# B&R Automation Studio project NAEUL004C00R13L518F00 (part 17)

#### Act_OptP0928MagConv1BtmFB.st
```iecst
ACTION Act_OptP0928MagConv1BtmFB:

	//Magazine Conveyor
	IF tyP0928MagConv.tyBtmFB.tyBtnStop.bRtCompl = TRUE THEN
		eOutMagConvAct	:= MagConvActStop;

		IF p_eOutMagConvStat = MagConvActStop AND p_eOutMagConvStatus = Done THEN
			eOutMagConvAct	:= MagConvActIdle;

			tyP0928MagConv.tyBtmFB.tyBtnEnt.bRtCompl	:= FALSE;
			tyP0928MagConv.tyBtmFB.tyBtnEnt.bValue		:= FALSE;
			tyP0928MagConv.tyBtmFB.tyBtnEnt.bRtLk		:= FALSE;

			tyP0928MagConv.tyBtmFB.tyBtnExit.bRtCompl	:= FALSE;
			tyP0928MagConv.tyBtmFB.tyBtnExit.bValue		:= FALSE;
			tyP0928MagConv.tyBtmFB.tyBtnExit.bRtLk		:= FALSE;

			tyP0928MagConv.tyBtmFB.tyBtnStop.bRtCompl	:= FALSE;
			tyP0928MagConv.tyBtmFB.tyBtnStop.bValue		:= TRUE;
			tyP0928MagConv.tyBtmFB.tyBtnStop.bRtLk		:= TRUE;
		END_IF

	ELSIF tyP0928MagConv.tyBtmFB.tyBtnEnt.bRtCompl = TRUE THEN
		tyP0928MagConv.tyBtmFB.tyBtnEnt.bValue	:= TRUE;
		tyP0928MagConv.tyBtmFB.tyBtnEnt.bRtLk		:= TRUE;

		tyP0928MagConv.tyBtmFB.tyBtnStop.bValue	:= FALSE;
		tyP0928MagConv.tyBtmFB.tyBtnStop.bRtLk	:= FALSE;

		eOutMagConvAct	:= MagConvActEnt;

		IF p_eOutMagConvStat = MagConvActEnt AND p_eOutMagConvStatus = Done THEN
			eOutMagConvAct	:= MagConvActIdle;

			tyP0928MagConv.tyBtmFB.tyBtnEnt.bRtCompl	:= FALSE;

			tyP0928MagConv.tyBtmFB.tyBtnEnt.bValue	:= FALSE;
			tyP0928MagConv.tyBtmFB.tyBtnEnt.bRtLk		:= FALSE;

			tyP0928MagConv.tyBtmFB.tyBtnStop.bValue	:= TRUE;
			tyP0928MagConv.tyBtmFB.tyBtnStop.bRtLk	:= TRUE;
		END_IF

	ELSIF tyP0928MagConv.tyBtmFB.tyBtnExit.bRtCompl = TRUE THEN
		tyP0928MagConv.tyBtmFB.tyBtnExit.bValue	:= TRUE;
		tyP0928MagConv.tyBtmFB.tyBtnExit.bRtLk	:= TRUE;

		tyP0928MagConv.tyBtmFB.tyBtnStop.bValue	:= FALSE;
		tyP0928MagConv.tyBtmFB.tyBtnStop.bRtLk	:= FALSE;

		eOutMagConvAct	:= MagConvActExit;

		IF p_eOutMagConvStat = MagConvActExit AND p_eOutMagConvStatus = Done THEN
			eOutMagConvAct	:= MagConvActIdle;

			tyP0928MagConv.tyBtmFB.tyBtnExit.bRtCompl:= FALSE;

			tyP0928MagConv.tyBtmFB.tyBtnExit.bValue	:= FALSE;
			tyP0928MagConv.tyBtmFB.tyBtnExit.bRtLk	:= FALSE;

			tyP0928MagConv.tyBtmFB.tyBtnStop.bValue	:= TRUE;
			tyP0928MagConv.tyBtmFB.tyBtnStop.bRtLk	:= TRUE;
		END_IF
	END_IF

	//Stopper
	IF tyP0928MagConv.tyCom.tyBtnSwitch.bValue = FALSE THEN

		//Mid stopper
		IF tyP0928MagConv.tyBtmFB.tyBtnMidStprExt.bRtCompl = TRUE THEN
			tyP0928MagConv.tyBtmFB.tyBtnMidStprExt.bRtCompl	:= FALSE;

			tyP0928MagConv.tyBtmFB.tyBtnMidStprExt.bValue	:= TRUE;
			tyP0928MagConv.tyBtmFB.tyBtnMidStprRet.bValue	:= FALSE;

		ELSIF tyP0928MagConv.tyBtmFB.tyBtnMidStprRet.bRtCompl = TRUE THEN
			tyP0928MagConv.tyBtmFB.tyBtnMidStprRet.bRtCompl	:= FALSE;

			tyP0928MagConv.tyBtmFB.tyBtnMidStprRet.bValue	:= TRUE;
			tyP0928MagConv.tyBtmFB.tyBtnMidStprExt.bValue	:= FALSE;

		END_IF

		//Ext Stopper
		IF tyP0928MagConv.tyBtmFB.tyBtnExtStprExt.bRtCompl = TRUE THEN
			tyP0928MagConv.tyBtmFB.tyBtnExtStprExt.bRtCompl	:= FALSE;

			tyP0928MagConv.tyBtmFB.tyBtnExtStprExt.bValue	:= TRUE;
			tyP0928MagConv.tyBtmFB.tyBtnExtStprRet.bValue	:= FALSE;

		ELSIF tyP0928MagConv.tyBtmFB.tyBtnExtStprRet.bRtCompl = TRUE THEN
			tyP0928MagConv.tyBtmFB.tyBtnExtStprRet.bRtCompl	:= FALSE;

			tyP0928MagConv.tyBtmFB.tyBtnExtStprRet.bValue	:= TRUE;
			tyP0928MagConv.tyBtmFB.tyBtnExtStprExt.bValue	:= FALSE;

		END_IF

		//Action------------

		IF tyP0928MagConv.tyBtmFB.tyBtnMidStprExt.bValue = TRUE THEN
				eStopper4Act	:= PneuActExt;

				IF p_eStopper4Stat = PneuActExt AND p_eStopper4Status = Done THEN
					eStopper4Act	:= PneuActIdle;
					tyP0928MagConv.tyBtmFB.tyBtnMidStprExt.bValue	:= FALSE;
				ELSIF p_eStopper4Status = Error THEN
					tyP0928MagConv.tyBtmFB.tyBtnMidStprExt.bValue	:= FALSE;
				END_IF

		ELSIF tyP0928MagConv.tyBtmFB.tyBtnMidStprRet.bValue = TRUE THEN
			eStopper4Act	:= PneuActRet;

			IF p_eStopper4Stat = PneuActRet AND p_eStopper4Status = Done THEN
				eStopper4Act	:= PneuActIdle;
				tyP0928MagConv.tyBtmFB.tyBtnMidStprRet.bValue := FALSE;
			ELSIF p_eStopper4Status = Error THEN
				tyP0928MagConv.tyBtmFB.tyBtnMidStprRet.bValue := FALSE;
			END_IF

		END_IF

		IF tyP0928MagConv.tyBtmFB.tyBtnExtStprExt.bValue = TRUE THEN
			eStopper5Act	:= PneuActExt;

			IF p_eStopper5Stat = PneuActExt AND p_eStopper5Status = Done THEN
				eStopper5Act	:= PneuActIdle;
				tyP0928MagConv.tyBtmFB.tyBtnExtStprExt.bValue	:= FALSE;
			ELSIF p_eStopper5Status = Error THEN
				tyP0928MagConv.tyBtmFB.tyBtnExtStprExt.bValue	:= FALSE;
			END_IF

		ELSIF tyP0928MagConv.tyBtmFB.tyBtnExtStprRet.bValue = TRUE THEN
			eStopper5Act	:= PneuActRet;

			IF p_eStopper5Stat = PneuActRet AND p_eStopper5Status = Done THEN
				eStopper5Act	:= PneuActIdle;
				tyP0928MagConv.tyBtmFB.tyBtnExtStprRet.bValue := FALSE;
			ELSIF p_eStopper5Status = Error THEN
				tyP0928MagConv.tyBtmFB.tyBtnExtStprRet.bValue := FALSE;
			END_IF

		END_IF

		//Update Status
//		tyP0930MagConvBtm1.tyDC.tyBtnFixedUnclamp.bValue	:= NOT p_bMagConvBtm2Clp1ClprFixClampCtrl;
//		tyP0930MagConvBtm1.tyDC.tyBtnFixedClamp.bValue		:= p_bMagConvBtm2Clp1ClprFixClampCtrl;
//		tyP0930MagConvBtm1.tyDC.tyBtnRemoteUnclamp.bValue	:= NOT p_bMagConvBtm2Clp1ClprRmtClampCtrl;
//		tyP0930MagConvBtm1.tyDC.tyBtnRemoteClamp.bValue	:= p_bMagConvBtm2Clp1ClprRmtClampCtrl;
//
//		tyP0930MagConvBtm1.tyDC.tyBtnSelUnclamp.bRtCompl	:= FALSE;
//		tyP0930MagConvBtm1.tyDC.tyBtnSelClamp.bRtCompl		:= FALSE;
//		tyP0930MagConvBtm1.tyDC.tyBtnSelUnclamp.bValue	:= p_bSelClamp1RetCtrl;
//		tyP0930MagConvBtm1.tyDC.tyBtnSelClamp.bValue	:= p_bSelClamp1ExtCtrl;
	END_IF

	//Mask
//	IF p_tyUsrMgmtCurrAccessRgt.bManualFBOnly THEN
//
//		fUIInRtStatOff(ADR(tyP0930MagConvBtm1.tyCom.tyBtnSwitch.uiMaskRtStat));
//
//	ELSE
//
//	IF p_eMagConvBtm2Clp1Status = Error THEN
//
//		fUIInRtStatOff(ADR(tyP0930MagConvBtm1.tyFB.tyBtnEnt.uiMaskRtStat));
//		fUIInRtStatOff(ADR(tyP0930MagConvBtm1.tyFB.tyBtnExit.uiMaskRtStat));
//		fUIInRtStatOff(ADR(tyP0930MagConvBtm1.tyFB.tyBtnFixedClamp.uiMaskRtStat));
//		fUIInRtStatOff(ADR(tyP0930MagConvBtm1.tyFB.tyBtnFixedUnclamp.uiMaskRtStat));
//		fUIInRtStatOff(ADR(tyP0930MagConvBtm1.tyFB.tyBtnRemoteClamp.uiMaskRtStat));
//		fUIInRtStatOff(ADR(tyP0930MagConvBtm1.tyFB.tyBtnRemoteUnclamp.uiMaskRtStat));
//		fUIInRtStatOff(ADR(tyP0930MagConvBtm1.tyFB.tyBtnSelClamp.uiMaskRtStat));
//		fUIInRtStatOff(ADR(tyP0930MagConvBtm1.tyFB.tyBtnSelUnclamp.uiMaskRtStat));
//		fUIInRtStatHide(ADR(tyP0930MagConvBtm1.tyCom.tyBtnSwitch.uiMaskRtStat));
//
//	ELSIF tyP0930MagConvBtm1.tyFB.tyBtnEnt.bRtCompl = TRUE THEN
//
//		fUIInRtStatHide(ADR(tyP0930MagConvBtm1.tyFB.tyBtnEnt.uiMaskRtStat));
//		fUIInRtStatOff(ADR(tyP0930MagConvBtm1.tyFB.tyBtnExit.uiMaskRtStat));
//		fUIInRtStatOff(ADR(tyP0930MagConvBtm1.tyFB.tyBtnFixedClamp.uiMaskRtStat));
//		fUIInRtStatOff(ADR(tyP0930MagConvBtm1.tyFB.tyBtnFixedUnclamp.uiMaskRtStat));
//		fUIInRtStatOff(ADR(tyP0930MagConvBtm1.tyFB.tyBtnRemoteClamp.uiMaskRtStat));
//		fUIInRtStatOff(ADR(tyP0930MagConvBtm1.tyFB.tyBtnRemoteUnclamp.uiMaskRtStat));
//		fUIInRtStatOff(ADR(tyP0930MagConvBtm1.tyFB.tyBtnSelClamp.uiMaskRtStat));
//		fUIInRtStatOff(ADR(tyP0930MagConvBtm1.tyFB.tyBtnSelUnclamp.uiMaskRtStat));
//		fUIInRtStatOff(ADR(tyP0930MagConvBtm1.tyCom.tyBtnSwitch.uiMaskRtStat));
//
//	ELSIF tyP0930MagConvBtm1.tyFB.tyBtnExit.bRtCompl = TRUE THEN
//
//			fUIInRtStatOff(ADR(tyP0930MagConvBtm1.tyFB.tyBtnEnt.uiMaskRtStat));
//		fUIInRtStatHide(ADR(tyP0930MagConvBtm1.tyFB.tyBtnExit.uiMaskRtStat));
//		fUIInRtStatOff(ADR(tyP0930MagConvBtm1.tyFB.tyBtnFixedClamp.uiMaskRtStat));
//		fUIInRtStatOff(ADR(tyP0930MagConvBtm1.tyFB.tyBtnFixedUnclamp.uiMaskRtStat));
//		fUIInRtStatOff(ADR(tyP0930MagConvBtm1.tyFB.tyBtnRemoteClamp.uiMaskRtStat));
//		fUIInRtStatOff(ADR(tyP0930MagConvBtm1.tyFB.tyBtnRemoteUnclamp.uiMaskRtStat));
//		fUIInRtStatOff(ADR(tyP0930MagConvBtm1.tyFB.tyBtnSelClamp.uiMaskRtStat));
//		fUIInRtStatOff(ADR(tyP0930MagConvBtm1.tyFB.tyBtnSelUnclamp.uiMaskRtStat));
//		fUIInRtStatOff(ADR(tyP0930MagConvBtm1.tyCom.tyBtnSwitch.uiMaskRtStat));
//
//	ELSIF tyP0930MagConvBtm1.tyFB.tyBtnFixedClamp.bValue = TRUE OR tyP0930MagConvBtm1.tyFB.tyBtnRemoteClamp.bValue = TRUE
//			OR tyP0930MagConvBtm1.tyFB.tyBtnFixedUnclamp.bValue = TRUE OR tyP0930MagConvBtm1.tyFB.tyBtnRemoteUnclamp.bValue = TRUE
//			OR tyP0930MagConvBtm1.tyFB.tyBtnSelUnclamp.bValue = TRUE OR tyP0930MagConvBtm1.tyFB.tyBtnSelClamp.bValue = TRUE
//			THEN
//
//		fUIInRtStatOff(ADR(tyP0930MagConvBtm1.tyFB.tyBtnEnt.uiMaskRtStat));
//		fUIInRtStatOff(ADR(tyP0930MagConvBtm1.tyFB.tyBtnExit.uiMaskRtStat));
//		fUIInRtStatHide(ADR(tyP0930MagConvBtm1.tyFB.tyBtnFixedClamp.uiMaskRtStat));
//		fUIInRtStatHide(ADR(tyP0930MagConvBtm1.tyFB.tyBtnFixedUnclamp.uiMaskRtStat));
//		fUIInRtStatHide(ADR(tyP0930MagConvBtm1.tyFB.tyBtnRemoteClamp.uiMaskRtStat));
//		fUIInRtStatHide(ADR(tyP0930MagConvBtm1.tyFB.tyBtnRemoteUnclamp.uiMaskRtStat));
//		fUIInRtStatHide(ADR(tyP0930MagConvBtm1.tyFB.tyBtnSelClamp.uiMaskRtStat));
//		fUIInRtStatHide(ADR(tyP0930MagConvBtm1.tyFB.tyBtnSelUnclamp.uiMaskRtStat));
//		fUIInRtStatOff(ADR(tyP0930MagConvBtm1.tyCom.tyBtnSwitch.uiMaskRtStat));
//
//	ELSE
//
//		fUIInRtStatHide(ADR(tyP0930MagConvBtm1.tyFB.tyBtnEnt.uiMaskRtStat));
//		fUIInRtStatHide(ADR(tyP0930MagConvBtm1.tyFB.tyBtnExit.uiMaskRtStat));
//		fUIInRtStatHide(ADR(tyP0930MagConvBtm1.tyFB.tyBtnFixedClamp.uiMaskRtStat));
//		fUIInRtStatHide(ADR(tyP0930MagConvBtm1.tyFB.tyBtnFixedUnclamp.uiMaskRtStat));
//		fUIInRtStatHide(ADR(tyP0930MagConvBtm1.tyFB.tyBtnRemoteClamp.uiMaskRtStat));
//		fUIInRtStatHide(ADR(tyP0930MagConvBtm1.tyFB.tyBtnRemoteUnclamp.uiMaskRtStat));
//		fUIInRtStatHide(ADR(tyP0930MagConvBtm1.tyFB.tyBtnSelClamp.uiMaskRtStat));
//		fUIInRtStatHide(ADR(tyP0930MagConvBtm1.tyFB.tyBtnSelUnclamp.uiMaskRtStat));
//		fUIInRtStatHide(ADR(tyP0930MagConvBtm1.tyCom.tyBtnSwitch.uiMaskRtStat));
//
//	END_IF
//END_IF
//
//	IF p_tyDI.bMagConvBtmCAB717MagSen1 THEN
//			fUIInRtStatOff(ADR(tyP0930MagConvBtm1.tyFB.tyBtnSelClamp.uiMaskRtStat));
//	END_IF
//
//	IF p_bMagConvBtm2Clp1ClprFixClampCtrl OR p_bMagConvBtm2Clp1ClprRmtClampCtrl THEN
//		fUIInRtStatOff(ADR(tyP0930MagConvBtm1.tyFB.tyBtnEnt.uiMaskRtStat));
//		fUIInRtStatOff(ADR(tyP0930MagConvBtm1.tyFB.tyBtnExit.uiMaskRtStat));
//	END_IF
//

END_ACTION
```

#### Act_OptP0928MagConv1TopDC.st
```iecst
ACTION Act_OptP0928MagConv1TopDC:

	//Magazine Conveyor
	IF tyP0928MagConv.tyTopDC.tyBtnStop.bRtCompl = TRUE THEN
		eInMagConvAct	:= MagConvActStop;

		IF p_eInMagConvStat = MagConvActStop AND p_eInMagConvStatus = Done THEN
			eInMagConvAct	:= MagConvActIdle;

			tyP0928MagConv.tyTopDC.tyBtnStop.bRtCompl		:= FALSE;
			tyP0928MagConv.tyTopDC.tyBtnStop.bValue		:= TRUE;
			tyP0928MagConv.tyTopDC.tyBtnStop.bRtLk		:= TRUE;

			tyP0928MagConv.tyTopDC.tyBtnMagIn.bRtCompl	:= FALSE;
			tyP0928MagConv.tyTopDC.tyBtnMagIn.bValue		:= FALSE;
			tyP0928MagConv.tyTopDC.tyBtnMagIn.bRtLk		:= FALSE;

			tyP0928MagConv.tyTopDC.tyBtnMagOut.bRtCompl	:= FALSE;
			tyP0928MagConv.tyTopDC.tyBtnMagOut.bValue		:= FALSE;
			tyP0928MagConv.tyTopDC.tyBtnMagOut.bRtLk		:= FALSE;
		END_IF

	ELSIF tyP0928MagConv.tyTopDC.tyBtnMagIn.bRtCompl = TRUE THEN
		tyP0928MagConv.tyTopDC.tyBtnMagIn.bValue	:= TRUE;
		tyP0928MagConv.tyTopDC.tyBtnMagIn.bRtLk	:= TRUE;

		tyP0928MagConv.tyTopDC.tyBtnStop.bValue	:= FALSE;
		tyP0928MagConv.tyTopDC.tyBtnStop.bRtLk	:= FALSE;

		IF p_tyNtParamCurr.eProjInMagConvDir = ConvDirLToR OR p_tyNtParamCurr.eProjInMagConvDir = ConvDirLToL THEN

			eInMagConvAct	:= MagConvActSetMtrSigOnOrLToR;

			IF p_eInMagConvStat = MagConvActSetMtrSigOnOrLToR AND p_eInMagConvStatus = Done THEN
				eInMagConvAct	:= MagConvActIdle;

				tyP0928MagConv.tyTopDC.tyBtnMagIn.bRtCompl	:= FALSE;
			END_IF

		ELSE

			eInMagConvAct	:= MagConvActSetMtrDirOrRToL;

			IF p_eInMagConvStat = MagConvActSetMtrDirOrRToL AND p_eInMagConvStatus = Done THEN
				eInMagConvAct	:= MagConvActIdle;

				tyP0928MagConv.tyTopDC.tyBtnMagIn.bRtCompl	:= FALSE;
			END_IF

		END_IF

	ELSIF tyP0928MagConv.tyTopDC.tyBtnMagOut.bRtCompl = TRUE THEN
		tyP0928MagConv.tyTopDC.tyBtnMagOut.bValue	:= TRUE;
		tyP0928MagConv.tyTopDC.tyBtnMagOut.bRtLk	:= TRUE;

		tyP0928MagConv.tyTopDC.tyBtnStop.bValue	:= FALSE;
		tyP0928MagConv.tyTopDC.tyBtnStop.bRtLk	:= FALSE;

		IF p_tyNtParamCurr.eProjMagConvDir = ConvDirLToR OR p_tyNtParamCurr.eProjInMagConvDir = ConvDirRToR THEN

			eInMagConvAct	:= MagConvActSetMtrSigOnOrLToR;

			IF p_eInMagConvStat = MagConvActSetMtrSigOnOrLToR AND p_eInMagConvStatus = Done THEN
				eInMagConvAct	:= MagConvActIdle;

				tyP0928MagConv.tyTopDC.tyBtnMagOut.bRtCompl	:= FALSE;
			END_IF

		ELSE

			eInMagConvAct	:= MagConvActSetMtrDirOrRToL;

			IF p_eInMagConvStat = MagConvActSetMtrDirOrRToL AND p_eInMagConvStatus = Done THEN
				eInMagConvAct	:= MagConvActIdle;

				tyP0928MagConv.tyTopDC.tyBtnMagOut.bRtCompl	:= FALSE;
			END_IF

		END_IF

	END_IF

	IF tyP0928MagConv.tyCom.tyBtnSwitch.bValue = TRUE THEN
		//Mag Conv Stopper1
		IF p_bStopper1TwoCtrlOut = FALSE THEN
			IF tyP0928MagConv.tyTopDC.tyBtnEntStprExt.bRtCompl = TRUE THEN
				tyP0928MagConv.tyTopDC.tyBtnEntStprExt.bValue := TRUE;
				tyP0928MagConv.tyTopDC.tyBtnEntStprRet.bValue := FALSE;

				eStopper1Act	:= PneuActSetExt;

				IF p_eStopper1Stat = PneuActSetExt AND p_eStopper1Status = Done THEN
					eStopper1Act	:= PneuActIdle;

					tyP0928MagConv.tyTopDC.tyBtnEntStprExt.bRtCompl	:= FALSE;
				END_IF

			ELSIF tyP0928MagConv.tyTopDC.tyBtnEntStprRet.bRtCompl = TRUE THEN
				tyP0928MagConv.tyTopDC.tyBtnEntStprRet.bValue := TRUE;
				tyP0928MagConv.tyTopDC.tyBtnEntStprExt.bValue := FALSE;

				eStopper1Act	:= PneuActSetRet;

				IF p_eStopper1Stat = PneuActSetRet AND p_eStopper1Status = Done THEN
					eStopper1Act	:= PneuActIdle;

					tyP0928MagConv.tyTopDC.tyBtnEntStprRet.bRtCompl	:= FALSE;
				END_IF
			END_IF

		ELSE
			IF (tyP0928MagConv.tyTopDC.tyBtnEntStprExt.bRtCompl = TRUE) OR (tyP0928MagConv.tyTopDC.tyBtnEntStprRet.bRtCompl = TRUE) THEN
				IF (tyP0928MagConv.tyTopDC.tyBtnEntStprExt.bValue = TRUE) AND (tyP0928MagConv.tyTopDC.tyBtnEntStprRet.bValue = TRUE) THEN
					eStopper1Act	:= PneuActSetAll;

					IF p_eStopper1Stat = PneuActSetAll AND p_eStopper1Status = Done THEN
						eStopper1Act	:= PneuActIdle;

						tyP0928MagConv.tyTopDC.tyBtnEntStprExt.bRtCompl		:= FALSE;
						tyP0928MagConv.tyTopDC.tyBtnEntStprRet.bRtCompl			:= FALSE;
					END_IF
					/////////i edited the ret to ext
				ELSIF (tyP0928MagConv.tyTopDC.tyBtnEntStprExt.bValue = TRUE) AND (tyP0928MagConv.tyTopDC.tyBtnEntStprRet.bValue = FALSE) THEN
					eStopper1Act	:= PneuActSetExt;(**)

					IF p_eStopper1Stat = PneuActSetExt (**) AND p_eStopper1Status = Done THEN
						eStopper1Act	:= PneuActIdle;

						tyP0928MagConv.tyTopDC.tyBtnEntStprExt.bRtCompl		:= FALSE;
						tyP0928MagConv.tyTopDC.tyBtnEntStprRet.bRtCompl		:= FALSE;
					END_IF

				ELSIF (tyP0928MagConv.tyTopDC.tyBtnEntStprExt.bValue = FALSE) AND (tyP0928MagConv.tyTopDC.tyBtnEntStprRet.bValue = TRUE) THEN
					eStopper1Act	:= PneuActSetRet;

					IF p_eStopper1Stat = PneuActSetRet AND p_eStopper1Status = Done THEN
						eStopper1Act	:= PneuActIdle;

						tyP0928MagConv.tyTopDC.tyBtnEntStprExt.bRtCompl		:= FALSE;
						tyP0928MagConv.tyTopDC.tyBtnEntStprRet.bRtCompl			:= FALSE;
					END_IF
					///////
				ELSE
					eStopper1Act	:= PneuActRstAll;

					IF p_eStopper1Stat = PneuActRstAll AND p_eStopper1Status = Done THEN
						eStopper1Act	:= PneuActIdle;

						tyP0928MagConv.tyTopDC.tyBtnEntStprExt.bRtCompl		:= FALSE;
						tyP0928MagConv.tyTopDC.tyBtnEntStprRet.bRtCompl			:= FALSE;
					END_IF

				END_IF
			END_IF
		END_IF//stopper1

		//Mag Conv Stopper2
		IF p_bStopper2TwoCtrlOut = FALSE THEN
			IF tyP0928MagConv.tyTopDC.tyBtnMidStprExt.bRtCompl = TRUE THEN
				tyP0928MagConv.tyTopDC.tyBtnMidStprExt.bValue := TRUE;
				tyP0928MagConv.tyTopDC.tyBtnMidStprRet.bValue := FALSE;

				eStopper2Act	:= PneuActSetExt;

				IF p_eStopper2Stat = PneuActSetExt AND p_eStopper2Status = Done THEN
					eStopper2Act	:= PneuActIdle;

					tyP0928MagConv.tyTopDC.tyBtnMidStprExt.bRtCompl	:= FALSE;
				END_IF

			ELSIF tyP0928MagConv.tyTopDC.tyBtnMidStprRet.bRtCompl = TRUE THEN
				tyP0928MagConv.tyTopDC.tyBtnMidStprRet.bValue := TRUE;
				tyP0928MagConv.tyTopDC.tyBtnMidStprExt.bValue := FALSE;

				eStopper2Act	:= PneuActSetRet;

				IF p_eStopper2Stat = PneuActSetRet AND p_eStopper2Status = Done THEN
					eStopper2Act	:= PneuActIdle;

					tyP0928MagConv.tyTopDC.tyBtnMidStprRet.bRtCompl	:= FALSE;
				END_IF
			END_IF

		ELSE
			IF (tyP0928MagConv.tyTopDC.tyBtnMidStprExt.bRtCompl = TRUE) OR (tyP0928MagConv.tyTopDC.tyBtnMidStprRet.bRtCompl = TRUE) THEN
				IF (tyP0928MagConv.tyTopDC.tyBtnMidStprExt.bValue = TRUE) AND (tyP0928MagConv.tyTopDC.tyBtnMidStprRet.bValue = TRUE) THEN
					eStopper2Act	:= PneuActSetAll;

					IF p_eStopper2Stat = PneuActSetAll AND p_eStopper2Status = Done THEN
						eStopper2Act	:= PneuActIdle;

						tyP0928MagConv.tyTopDC.tyBtnMidStprExt.bRtCompl		:= FALSE;
						tyP0928MagConv.tyTopDC.tyBtnMidStprRet.bRtCompl			:= FALSE;
					END_IF
					/////////i edited the ret to ext
				ELSIF (tyP0928MagConv.tyTopDC.tyBtnMidStprExt.bValue = TRUE) AND (tyP0928MagConv.tyTopDC.tyBtnMidStprRet.bValue = FALSE) THEN
					eStopper2Act	:= PneuActSetExt;(**)

					IF p_eStopper2Stat = PneuActSetExt (**) AND p_eStopper2Status = Done THEN
						eStopper2Act	:= PneuActIdle;

						tyP0928MagConv.tyTopDC.tyBtnMidStprExt.bRtCompl		:= FALSE;
						tyP0928MagConv.tyTopDC.tyBtnMidStprRet.bRtCompl		:= FALSE;
					END_IF

				ELSIF (tyP0928MagConv.tyTopDC.tyBtnMidStprExt.bValue = FALSE) AND (tyP0928MagConv.tyTopDC.tyBtnMidStprRet.bValue = TRUE) THEN
					eStopper2Act	:= PneuActSetRet;

					IF p_eStopper2Stat = PneuActSetRet AND p_eStopper2Status = Done THEN
						eStopper2Act	:= PneuActIdle;

						tyP0928MagConv.tyTopDC.tyBtnMidStprExt.bRtCompl		:= FALSE;
						tyP0928MagConv.tyTopDC.tyBtnMidStprRet.bRtCompl			:= FALSE;
					END_IF
					///////
				ELSE
					eStopper2Act	:= PneuActRstAll;

					IF p_eStopper2Stat = PneuActRstAll AND p_eStopper2Status = Done THEN
						eStopper2Act	:= PneuActIdle;

						tyP0928MagConv.tyTopDC.tyBtnMidStprExt.bRtCompl		:= FALSE;
						tyP0928MagConv.tyTopDC.tyBtnMidStprRet.bRtCompl			:= FALSE;
					END_IF

				END_IF
			END_IF
		END_IF//stopper2

		//Mag Conv Stopper3
		IF p_bStopper3TwoCtrlOut = FALSE THEN
			IF tyP0928MagConv.tyTopDC.tyBtnExtStprExt.bRtCompl = TRUE THEN
				tyP0928MagConv.tyTopDC.tyBtnExtStprExt.bValue := TRUE;
				tyP0928MagConv.tyTopDC.tyBtnExtStprRet.bValue := FALSE;

				eStopper3Act	:= PneuActSetExt;

				IF p_eStopper3Stat = PneuActSetExt AND p_eStopper3Status = Done THEN
					eStopper3Act	:= PneuActIdle;

					tyP0928MagConv.tyTopDC.tyBtnExtStprExt.bRtCompl	:= FALSE;
				END_IF

			ELSIF tyP0928MagConv.tyTopDC.tyBtnExtStprRet.bRtCompl = TRUE THEN
				tyP0928MagConv.tyTopDC.tyBtnExtStprRet.bValue := TRUE;
				tyP0928MagConv.tyTopDC.tyBtnExtStprExt.bValue := FALSE;

				eStopper3Act	:= PneuActSetRet;

				IF p_eStopper3Stat = PneuActSetRet AND p_eStopper3Status = Done THEN
					eStopper3Act	:= PneuActIdle;

					tyP0928MagConv.tyTopDC.tyBtnExtStprRet.bRtCompl	:= FALSE;
				END_IF
			END_IF

		ELSE
			IF (tyP0928MagConv.tyTopDC.tyBtnExtStprExt.bRtCompl = TRUE) OR (tyP0928MagConv.tyTopDC.tyBtnExtStprRet.bRtCompl = TRUE) THEN
				IF (tyP0928MagConv.tyTopDC.tyBtnExtStprExt.bValue = TRUE) AND (tyP0928MagConv.tyTopDC.tyBtnExtStprRet.bValue = TRUE) THEN
					eStopper3Act	:= PneuActSetAll;

					IF p_eStopper3Stat = PneuActSetAll AND p_eStopper3Status = Done THEN
						eStopper3Act	:= PneuActIdle;

						tyP0928MagConv.tyTopDC.tyBtnExtStprExt.bRtCompl		:= FALSE;
						tyP0928MagConv.tyTopDC.tyBtnExtStprRet.bRtCompl			:= FALSE;
					END_IF
					/////////i edited the ret to ext
				ELSIF (tyP0928MagConv.tyTopDC.tyBtnExtStprExt.bValue = TRUE) AND (tyP0928MagConv.tyTopDC.tyBtnExtStprRet.bValue = FALSE) THEN
					eStopper3Act	:= PneuActSetExt;(**)

					IF p_eStopper3Stat = PneuActSetExt (**) AND p_eStopper3Status = Done THEN
						eStopper3Act	:= PneuActIdle;

						tyP0928MagConv.tyTopDC.tyBtnExtStprExt.bRtCompl		:= FALSE;
						tyP0928MagConv.tyTopDC.tyBtnExtStprRet.bRtCompl		:= FALSE;
					END_IF

				ELSIF (tyP0928MagConv.tyTopDC.tyBtnExtStprExt.bValue = FALSE) AND (tyP0928MagConv.tyTopDC.tyBtnExtStprRet.bValue = TRUE) THEN
					eStopper3Act	:= PneuActSetRet;

					IF p_eStopper3Stat = PneuActSetRet AND p_eStopper3Status = Done THEN
						eStopper3Act	:= PneuActIdle;

						tyP0928MagConv.tyTopDC.tyBtnExtStprExt.bRtCompl		:= FALSE;
						tyP0928MagConv.tyTopDC.tyBtnExtStprRet.bRtCompl			:= FALSE;
					END_IF
					///////
				ELSE
					eStopper3Act	:= PneuActRstAll;

					IF p_eStopper3Stat = PneuActRstAll AND p_eStopper3Status = Done THEN
						eStopper3Act	:= PneuActIdle;

						tyP0928MagConv.tyTopDC.tyBtnExtStprExt.bRtCompl		:= FALSE;
						tyP0928MagConv.tyTopDC.tyBtnExtStprRet.bRtCompl			:= FALSE;
					END_IF

				END_IF
			END_IF
		END_IF//stopper3

		//ent
		tyP0928MagConv.tyTopFB.tyBtnEntStprExt.bRtCompl		:= FALSE;
		tyP0928MagConv.tyTopFB.tyBtnEntStprExt.bValue		:= FALSE;
		tyP0928MagConv.tyTopFB.tyBtnEntStprRet.bRtCompl		:= FALSE;
		tyP0928MagConv.tyTopFB.tyBtnEntStprRet.bValue		:= FALSE;

		//mid
		tyP0928MagConv.tyTopFB.tyBtnMidStprExt.bRtCompl		:= FALSE;
		tyP0928MagConv.tyTopFB.tyBtnMidStprExt.bValue		:= FALSE;
		tyP0928MagConv.tyTopFB.tyBtnMidStprRet.bRtCompl		:= FALSE;
		tyP0928MagConv.tyTopFB.tyBtnMidStprRet.bValue		:= FALSE;

		//ext
		tyP0928MagConv.tyTopFB.tyBtnExtStprExt.bRtCompl		:= FALSE;
		tyP0928MagConv.tyTopFB.tyBtnExtStprExt.bValue		:= FALSE;
		tyP0928MagConv.tyTopFB.tyBtnExtStprRet.bRtCompl		:= FALSE;
		tyP0928MagConv.tyTopFB.tyBtnExtStprRet.bValue		:= FALSE;
	END_IF

	//Mask
//	IF p_eInMagConvStatus = Error THEN
//
//		fUIInRtStatOff(ADR(tyP0928MagConv.tyTopDC.tyBtnMagIn.uiMaskRtStat));
//		fUIInRtStatOff(ADR(tyP0928MagConv.tyTopDC.tyBtnMagOut.uiMaskRtStat));
//		fUIInRtStatOff(ADR(tyP0928MagConv.tyTopDC.tyBtnFixedClamp.uiMaskRtStat));
//		fUIInRtStatOff(ADR(tyP0928MagConv.tyTopDC.tyBtnFixedUnclamp.uiMaskRtStat));
//		fUIInRtStatOff(ADR(tyP0928MagConv.tyTopDC.tyBtnRemoteClamp.uiMaskRtStat));
//		fUIInRtStatOff(ADR(tyP0928MagConv.tyTopDC.tyBtnRemoteUnclamp.uiMaskRtStat));
//		fUIInRtStatOff(ADR(tyP0928MagConv.tyTopDC.tyBtnSelClamp.uiMaskRtStat));
//		fUIInRtStatOff(ADR(tyP0928MagConv.tyTopDC.tyBtnSelUnclamp.uiMaskRtStat));
//
//	ELSIF tyP0928MagConv.tyTopDC.tyBtnMagIn.bValue = TRUE THEN
//
//		fUIInRtStatHide(ADR(tyP0928MagConv.tyTopDC.tyBtnMagIn.uiMaskRtStat));
//		fUIInRtStatOff(ADR(tyP0928MagConv.tyTopDC.tyBtnMagOut.uiMaskRtStat));
//		fUIInRtStatOff(ADR(tyP0928MagConv.tyTopDC.tyBtnFixedClamp.uiMaskRtStat));
//		fUIInRtStatOff(ADR(tyP0928MagConv.tyTopDC.tyBtnFixedUnclamp.uiMaskRtStat));
//		fUIInRtStatOff(ADR(tyP0928MagConv.tyTopDC.tyBtnRemoteClamp.uiMaskRtStat));
//		fUIInRtStatOff(ADR(tyP0928MagConv.tyTopDC.tyBtnRemoteUnclamp.uiMaskRtStat));
//		fUIInRtStatOff(ADR(tyP0928MagConv.tyTopDC.tyBtnSelClamp.uiMaskRtStat));
//		fUIInRtStatOff(ADR(tyP0928MagConv.tyTopDC.tyBtnSelUnclamp.uiMaskRtStat));
//
//	ELSIF tyP0928MagConv.tyTopDC.tyBtnMagOut.bValue = TRUE THEN
//
//		fUIInRtStatOff(ADR(tyP0928MagConv.tyTopDC.tyBtnMagIn.uiMaskRtStat));
//		fUIInRtStatHide(ADR(tyP0928MagConv.tyTopDC.tyBtnMagOut.uiMaskRtStat));
//		fUIInRtStatOff(ADR(tyP0928MagConv.tyTopDC.tyBtnFixedClamp.uiMaskRtStat));
//		fUIInRtStatOff(ADR(tyP0928MagConv.tyTopDC.tyBtnFixedUnclamp.uiMaskRtStat));
//		fUIInRtStatOff(ADR(tyP0928MagConv.tyTopDC.tyBtnRemoteClamp.uiMaskRtStat));
//		fUIInRtStatOff(ADR(tyP0928MagConv.tyTopDC.tyBtnRemoteUnclamp.uiMaskRtStat));
//		fUIInRtStatOff(ADR(tyP0928MagConv.tyTopDC.tyBtnSelClamp.uiMaskRtStat));
//		fUIInRtStatOff(ADR(tyP0928MagConv.tyTopDC.tyBtnSelUnclamp.uiMaskRtStat));
//
//	ELSE
//
//		fUIInRtStatHide(ADR(tyP0928MagConv.tyTopDC.tyBtnMagIn.uiMaskRtStat));
//		fUIInRtStatHide(ADR(tyP0928MagConv.tyTopDC.tyBtnMagOut.uiMaskRtStat));
//		fUIInRtStatHide(ADR(tyP0928MagConv.tyTopDC.tyBtnFixedClamp.uiMaskRtStat));
//		fUIInRtStatHide(ADR(tyP0928MagConv.tyTopDC.tyBtnFixedUnclamp.uiMaskRtStat));
//		fUIInRtStatHide(ADR(tyP0928MagConv.tyTopDC.tyBtnRemoteClamp.uiMaskRtStat));
//		fUIInRtStatHide(ADR(tyP0928MagConv.tyTopDC.tyBtnRemoteUnclamp.uiMaskRtStat));
//		fUIInRtStatHide(ADR(tyP0928MagConv.tyTopDC.tyBtnSelClamp.uiMaskRtStat));
//		fUIInRtStatHide(ADR(tyP0928MagConv.tyTopDC.tyBtnSelUnclamp.uiMaskRtStat));
//
//	END_IF
//

END_ACTION
```

#### Act_OptP0928MagConv1BtmDC.st
```iecst
ACTION Act_OptP0928MagConv1BtmDC:

	//Magazine Conveyor
	IF tyP0928MagConv.tyBtmDC.tyBtnStop.bRtCompl = TRUE THEN
		eOutMagConvAct	:= MagConvActStop;

		IF p_eOutMagConvStat = MagConvActStop AND p_eOutMagConvStatus = Done THEN
			eOutMagConvAct	:= MagConvActIdle;

			tyP0928MagConv.tyBtmDC.tyBtnStop.bRtCompl		:= FALSE;
			tyP0928MagConv.tyBtmDC.tyBtnStop.bValue		:= TRUE;
			tyP0928MagConv.tyBtmDC.tyBtnStop.bRtLk		:= TRUE;

			tyP0928MagConv.tyBtmDC.tyBtnMagIn.bRtCompl	:= FALSE;
			tyP0928MagConv.tyBtmDC.tyBtnMagIn.bValue		:= FALSE;
			tyP0928MagConv.tyBtmDC.tyBtnMagIn.bRtLk		:= FALSE;

			tyP0928MagConv.tyBtmDC.tyBtnMagOut.bRtCompl	:= FALSE;
			tyP0928MagConv.tyBtmDC.tyBtnMagOut.bValue		:= FALSE;
			tyP0928MagConv.tyBtmDC.tyBtnMagOut.bRtLk		:= FALSE;
		END_IF

	ELSIF tyP0928MagConv.tyBtmDC.tyBtnMagIn.bRtCompl = TRUE THEN
		tyP0928MagConv.tyBtmDC.tyBtnMagIn.bValue	:= TRUE;
		tyP0928MagConv.tyBtmDC.tyBtnMagIn.bRtLk	:= TRUE;

		tyP0928MagConv.tyBtmDC.tyBtnStop.bValue	:= FALSE;
		tyP0928MagConv.tyBtmDC.tyBtnStop.bRtLk	:= FALSE;

		IF p_tyNtParamCurr.eProjOutMagConvDir = ConvDirLToR OR p_tyNtParamCurr.eProjOutMagConvDir = ConvDirLToL THEN

			eOutMagConvAct	:= MagConvActSetMtrSigOnOrLToR;

			IF p_eOutMagConvStat = MagConvActSetMtrSigOnOrLToR AND p_eOutMagConvStatus = Done THEN
				eOutMagConvAct	:= MagConvActIdle;

				tyP0928MagConv.tyBtmDC.tyBtnMagIn.bRtCompl	:= FALSE;
			END_IF

		ELSE

			eOutMagConvAct	:= MagConvActSetMtrDirOrRToL;

			IF p_eOutMagConvStat = MagConvActSetMtrDirOrRToL AND p_eOutMagConvStatus = Done THEN
				eOutMagConvAct	:= MagConvActIdle;

				tyP0928MagConv.tyBtmDC.tyBtnMagIn.bRtCompl	:= FALSE;
			END_IF

		END_IF

	ELSIF tyP0928MagConv.tyBtmDC.tyBtnMagOut.bRtCompl = TRUE THEN
		tyP0928MagConv.tyBtmDC.tyBtnMagOut.bValue	:= TRUE;
		tyP0928MagConv.tyBtmDC.tyBtnMagOut.bRtLk	:= TRUE;

		tyP0928MagConv.tyBtmDC.tyBtnStop.bValue	:= FALSE;
		tyP0928MagConv.tyBtmDC.tyBtnStop.bRtLk	:= FALSE;

		IF p_tyNtParamCurr.eProjOutMagConvDir = ConvDirLToR OR p_tyNtParamCurr.eProjOutMagConvDir = ConvDirRToR THEN

			eOutMagConvAct	:= MagConvActSetMtrSigOnOrLToR;

			IF p_eOutMagConvStat = MagConvActSetMtrSigOnOrLToR AND p_eOutMagConvStatus = Done THEN
				eOutMagConvAct	:= MagConvActIdle;

				tyP0928MagConv.tyBtmDC.tyBtnMagOut.bRtCompl	:= FALSE;
			END_IF

		ELSE

			eOutMagConvAct	:= MagConvActSetMtrDirOrRToL;

			IF p_eOutMagConvStat = MagConvActSetMtrDirOrRToL AND p_eOutMagConvStatus = Done THEN
				eOutMagConvAct	:= MagConvActIdle;

				tyP0928MagConv.tyBtmDC.tyBtnMagOut.bRtCompl	:= FALSE;
			END_IF

		END_IF

	END_IF

	IF tyP0928MagConv.tyCom.tyBtnSwitch.bValue = TRUE THEN

		//Mag Conv Stopper4
		IF p_bStopper4TwoCtrlOut = FALSE THEN
			IF tyP0928MagConv.tyBtmDC.tyBtnMidStprExt.bRtCompl = TRUE THEN
				tyP0928MagConv.tyBtmDC.tyBtnMidStprExt.bValue := TRUE;
				tyP0928MagConv.tyBtmDC.tyBtnMidStprRet.bValue := FALSE;

				eStopper4Act	:= PneuActSetExt;

				IF p_eStopper4Stat = PneuActSetExt AND p_eStopper4Status = Done THEN
					eStopper4Act	:= PneuActIdle;

					tyP0928MagConv.tyBtmDC.tyBtnMidStprExt.bRtCompl	:= FALSE;
				END_IF

			ELSIF tyP0928MagConv.tyBtmDC.tyBtnMidStprRet.bRtCompl = TRUE THEN
				tyP0928MagConv.tyBtmDC.tyBtnMidStprRet.bValue := TRUE;
				tyP0928MagConv.tyBtmDC.tyBtnMidStprExt.bValue := FALSE;

				eStopper4Act	:= PneuActSetRet;

				IF p_eStopper4Stat = PneuActSetRet AND p_eStopper4Status = Done THEN
					eStopper4Act	:= PneuActIdle;

					tyP0928MagConv.tyBtmDC.tyBtnMidStprRet.bRtCompl	:= FALSE;
				END_IF
			END_IF

		ELSE
			IF (tyP0928MagConv.tyBtmDC.tyBtnMidStprExt.bRtCompl = TRUE) OR (tyP0928MagConv.tyBtmDC.tyBtnMidStprRet.bRtCompl = TRUE) THEN
				IF (tyP0928MagConv.tyBtmDC.tyBtnMidStprExt.bValue = TRUE) AND (tyP0928MagConv.tyBtmDC.tyBtnMidStprRet.bValue = TRUE) THEN
					eStopper4Act	:= PneuActSetAll;

					IF p_eStopper4Stat = PneuActSetAll AND p_eStopper4Status = Done THEN
						eStopper4Act	:= PneuActIdle;

						tyP0928MagConv.tyBtmDC.tyBtnMidStprExt.bRtCompl		:= FALSE;
						tyP0928MagConv.tyBtmDC.tyBtnMidStprRet.bRtCompl			:= FALSE;
					END_IF
					/////////i edited the ret to ext
				ELSIF (tyP0928MagConv.tyBtmDC.tyBtnMidStprExt.bValue = TRUE) AND (tyP0928MagConv.tyBtmDC.tyBtnMidStprRet.bValue = FALSE) THEN
					eStopper4Act	:= PneuActSetExt;(**)

					IF p_eStopper4Stat = PneuActSetExt (**) AND p_eStopper4Status = Done THEN
						eStopper4Act	:= PneuActIdle;

						tyP0928MagConv.tyBtmDC.tyBtnMidStprExt.bRtCompl		:= FALSE;
						tyP0928MagConv.tyBtmDC.tyBtnMidStprRet.bRtCompl		:= FALSE;
					END_IF

				ELSIF (tyP0928MagConv.tyBtmDC.tyBtnMidStprExt.bValue = FALSE) AND (tyP0928MagConv.tyBtmDC.tyBtnMidStprRet.bValue = TRUE) THEN
					eStopper4Act	:= PneuActSetRet;

					IF p_eStopper4Stat = PneuActSetRet AND p_eStopper4Status = Done THEN
						eStopper4Act	:= PneuActIdle;

						tyP0928MagConv.tyBtmDC.tyBtnMidStprExt.bRtCompl		:= FALSE;
						tyP0928MagConv.tyBtmDC.tyBtnMidStprRet.bRtCompl			:= FALSE;
					END_IF
					///////
				ELSE
					eStopper4Act	:= PneuActRstAll;

					IF p_eStopper4Stat = PneuActRstAll AND p_eStopper4Status = Done THEN
						eStopper4Act	:= PneuActIdle;

						tyP0928MagConv.tyBtmDC.tyBtnMidStprExt.bRtCompl		:= FALSE;
						tyP0928MagConv.tyBtmDC.tyBtnMidStprRet.bRtCompl			:= FALSE;
					END_IF

				END_IF
			END_IF
		END_IF//Stopper4

		//Mag Conv Stopper5
		IF p_bStopper5TwoCtrlOut = FALSE THEN
			IF tyP0928MagConv.tyBtmDC.tyBtnExtStprExt.bRtCompl = TRUE THEN
				tyP0928MagConv.tyBtmDC.tyBtnExtStprExt.bValue := TRUE;
				tyP0928MagConv.tyBtmDC.tyBtnExtStprRet.bValue := FALSE;

				eStopper5Act	:= PneuActSetExt;

				IF p_eStopper5Stat = PneuActSetExt AND p_eStopper5Status = Done THEN
					eStopper5Act	:= PneuActIdle;

					tyP0928MagConv.tyBtmDC.tyBtnExtStprExt.bRtCompl	:= FALSE;
				END_IF

			ELSIF tyP0928MagConv.tyBtmDC.tyBtnExtStprRet.bRtCompl = TRUE THEN
				tyP0928MagConv.tyBtmDC.tyBtnExtStprRet.bValue := TRUE;
				tyP0928MagConv.tyBtmDC.tyBtnExtStprExt.bValue := FALSE;

				eStopper5Act	:= PneuActSetRet;

				IF p_eStopper5Stat = PneuActSetRet AND p_eStopper5Status = Done THEN
					eStopper5Act	:= PneuActIdle;

					tyP0928MagConv.tyBtmDC.tyBtnExtStprRet.bRtCompl	:= FALSE;
				END_IF
			END_IF

		ELSE
			IF (tyP0928MagConv.tyBtmDC.tyBtnExtStprExt.bRtCompl = TRUE) OR (tyP0928MagConv.tyBtmDC.tyBtnExtStprRet.bRtCompl = TRUE) THEN
				IF (tyP0928MagConv.tyBtmDC.tyBtnExtStprExt.bValue = TRUE) AND (tyP0928MagConv.tyBtmDC.tyBtnExtStprRet.bValue = TRUE) THEN
					eStopper5Act	:= PneuActSetAll;

					IF p_eStopper5Stat = PneuActSetAll AND p_eStopper5Status = Done THEN
						eStopper5Act	:= PneuActIdle;

						tyP0928MagConv.tyBtmDC.tyBtnExtStprExt.bRtCompl		:= FALSE;
						tyP0928MagConv.tyBtmDC.tyBtnExtStprRet.bRtCompl			:= FALSE;
					END_IF
					/////////i edited the ret to ext
				ELSIF (tyP0928MagConv.tyBtmDC.tyBtnExtStprExt.bValue = TRUE) AND (tyP0928MagConv.tyBtmDC.tyBtnExtStprRet.bValue = FALSE) THEN
					eStopper5Act	:= PneuActSetExt;(**)

					IF p_eStopper5Stat = PneuActSetExt (**) AND p_eStopper5Status = Done THEN
						eStopper5Act	:= PneuActIdle;

						tyP0928MagConv.tyBtmDC.tyBtnExtStprExt.bRtCompl		:= FALSE;
						tyP0928MagConv.tyBtmDC.tyBtnExtStprRet.bRtCompl		:= FALSE;
					END_IF

				ELSIF (tyP0928MagConv.tyBtmDC.tyBtnExtStprExt.bValue = FALSE) AND (tyP0928MagConv.tyBtmDC.tyBtnExtStprRet.bValue = TRUE) THEN
					eStopper5Act	:= PneuActSetRet;

					IF p_eStopper5Stat = PneuActSetRet AND p_eStopper5Status = Done THEN
						eStopper5Act	:= PneuActIdle;

						tyP0928MagConv.tyBtmDC.tyBtnExtStprExt.bRtCompl		:= FALSE;
						tyP0928MagConv.tyBtmDC.tyBtnExtStprRet.bRtCompl			:= FALSE;
					END_IF
					///////
				ELSE
					eStopper5Act	:= PneuActRstAll;

					IF p_eStopper5Stat = PneuActRstAll AND p_eStopper5Status = Done THEN
						eStopper5Act	:= PneuActIdle;

						tyP0928MagConv.tyBtmDC.tyBtnExtStprExt.bRtCompl		:= FALSE;
						tyP0928MagConv.tyBtmDC.tyBtnExtStprRet.bRtCompl			:= FALSE;
					END_IF

				END_IF
			END_IF
		END_IF//Stopper5

		//mid
		tyP0928MagConv.tyBtmFB.tyBtnMidStprExt.bRtCompl		:= FALSE;
		tyP0928MagConv.tyBtmFB.tyBtnMidStprExt.bValue		:= FALSE;
		tyP0928MagConv.tyBtmFB.tyBtnMidStprRet.bRtCompl		:= FALSE;
		tyP0928MagConv.tyBtmFB.tyBtnMidStprRet.bValue		:= FALSE;

		//ext
		tyP0928MagConv.tyBtmFB.tyBtnExtStprExt.bRtCompl		:= FALSE;
		tyP0928MagConv.tyBtmFB.tyBtnExtStprExt.bValue		:= FALSE;
		tyP0928MagConv.tyBtmFB.tyBtnExtStprRet.bRtCompl		:= FALSE;
		tyP0928MagConv.tyBtmFB.tyBtnExtStprRet.bValue		:= FALSE;
	END_IF

	//Mask
//	IF p_eOutMagConvStatus = Error THEN
//
//		fUIInRtStatOff(ADR(tyP0928MagConv.tyBtmDC.tyBtnMagIn.uiMaskRtStat));
//		fUIInRtStatOff(ADR(tyP0928MagConv.tyBtmDC.tyBtnMagOut.uiMaskRtStat));
//		fUIInRtStatOff(ADR(tyP0928MagConv.tyBtmDC.tyBtnFixedClamp.uiMaskRtStat));
//		fUIInRtStatOff(ADR(tyP0928MagConv.tyBtmDC.tyBtnFixedUnclamp.uiMaskRtStat));
//		fUIInRtStatOff(ADR(tyP0928MagConv.tyBtmDC.tyBtnRemoteClamp.uiMaskRtStat));
//		fUIInRtStatOff(ADR(tyP0928MagConv.tyBtmDC.tyBtnRemoteUnclamp.uiMaskRtStat));
//		fUIInRtStatOff(ADR(tyP0928MagConv.tyBtmDC.tyBtnSelClamp.uiMaskRtStat));
//		fUIInRtStatOff(ADR(tyP0928MagConv.tyBtmDC.tyBtnSelUnclamp.uiMaskRtStat));
//
//	ELSIF tyP0928MagConv.tyBtmDC.tyBtnMagIn.bValue = TRUE THEN
//
//		fUIInRtStatHide(ADR(tyP0928MagConv.tyBtmDC.tyBtnMagIn.uiMaskRtStat));
//		fUIInRtStatOff(ADR(tyP0928MagConv.tyBtmDC.tyBtnMagOut.uiMaskRtStat));
//		fUIInRtStatOff(ADR(tyP0928MagConv.tyBtmDC.tyBtnFixedClamp.uiMaskRtStat));
//		fUIInRtStatOff(ADR(tyP0928MagConv.tyBtmDC.tyBtnFixedUnclamp.uiMaskRtStat));
//		fUIInRtStatOff(ADR(tyP0928MagConv.tyBtmDC.tyBtnRemoteClamp.uiMaskRtStat));
//		fUIInRtStatOff(ADR(tyP0928MagConv.tyBtmDC.tyBtnRemoteUnclamp.uiMaskRtStat));
//		fUIInRtStatOff(ADR(tyP0928MagConv.tyBtmDC.tyBtnSelClamp.uiMaskRtStat));
//		fUIInRtStatOff(ADR(tyP0928MagConv.tyBtmDC.tyBtnSelUnclamp.uiMaskRtStat));
//
//	ELSIF tyP0928MagConv.tyBtmDC.tyBtnMagOut.bValue = TRUE THEN
//
//		fUIInRtStatOff(ADR(tyP0928MagConv.tyBtmDC.tyBtnMagIn.uiMaskRtStat));
//		fUIInRtStatHide(ADR(tyP0928MagConv.tyBtmDC.tyBtnMagOut.uiMaskRtStat));
//		fUIInRtStatOff(ADR(tyP0928MagConv.tyBtmDC.tyBtnFixedClamp.uiMaskRtStat));
//		fUIInRtStatOff(ADR(tyP0928MagConv.tyBtmDC.tyBtnFixedUnclamp.uiMaskRtStat));
//		fUIInRtStatOff(ADR(tyP0928MagConv.tyBtmDC.tyBtnRemoteClamp.uiMaskRtStat));
//		fUIInRtStatOff(ADR(tyP0928MagConv.tyBtmDC.tyBtnRemoteUnclamp.uiMaskRtStat));
//		fUIInRtStatOff(ADR(tyP0928MagConv.tyBtmDC.tyBtnSelClamp.uiMaskRtStat));
//		fUIInRtStatOff(ADR(tyP0928MagConv.tyBtmDC.tyBtnSelUnclamp.uiMaskRtStat));
//
//	ELSE
//
//		fUIInRtStatHide(ADR(tyP0928MagConv.tyBtmDC.tyBtnMagIn.uiMaskRtStat));
//		fUIInRtStatHide(ADR(tyP0928MagConv.tyBtmDC.tyBtnMagOut.uiMaskRtStat));
//		fUIInRtStatHide(ADR(tyP0928MagConv.tyBtmDC.tyBtnFixedClamp.uiMaskRtStat));
//		fUIInRtStatHide(ADR(tyP0928MagConv.tyBtmDC.tyBtnFixedUnclamp.uiMaskRtStat));
//		fUIInRtStatHide(ADR(tyP0928MagConv.tyBtmDC.tyBtnRemoteClamp.uiMaskRtStat));
//		fUIInRtStatHide(ADR(tyP0928MagConv.tyBtmDC.tyBtnRemoteUnclamp.uiMaskRtStat));
//		fUIInRtStatHide(ADR(tyP0928MagConv.tyBtmDC.tyBtnSelClamp.uiMaskRtStat));
//		fUIInRtStatHide(ADR(tyP0928MagConv.tyBtmDC.tyBtnSelUnclamp.uiMaskRtStat));
//
//	END_IF
//

END_ACTION
```

#### Act_OptP0928RstMnlTop.st
```iecst
ACTION Act_OptP0928RstMnlTop:

	IF EDGEPOS((bManualMod = FALSE) OR (p_eInMagConvStatus = Error)) THEN

		eInMagConvAct	:= MagConvActIdle;
		//Magazine Conveyor
		//FB
		tyP0928MagConv.tyTopFB.tyBtnEnt.bRtCompl				:= FALSE;
		tyP0928MagConv.tyTopFB.tyBtnExit.bRtCompl				:= FALSE;
		tyP0928MagConv.tyTopFB.tyBtnStop.bRtCompl				:= FALSE;

		tyP0928MagConv.tyTopFB.tyBtnEnt.bValue				:= FALSE;
		tyP0928MagConv.tyTopFB.tyBtnExit.bValue				:= FALSE;
		tyP0928MagConv.tyTopFB.tyBtnStop.bValue				:= TRUE;

		tyP0928MagConv.tyTopFB.tyBtnEnt.bRtLk				:= FALSE;
		tyP0928MagConv.tyTopFB.tyBtnExit.bRtLk				:= FALSE;
		tyP0928MagConv.tyTopFB.tyBtnStop.bRtLk				:= TRUE;

		tyP0928MagConv.tyTopFB.tyBtnEnt.uiMaskRtStat.0		:= TRUE;
		tyP0928MagConv.tyTopFB.tyBtnExit.uiMaskRtStat.0		:= TRUE;
		tyP0928MagConv.tyCom.tyBtnSwitch.uiMaskRtStat.0		:= TRUE;

		//Direct
		tyP0928MagConv.tyTopDC.tyBtnMagIn.bRtCompl				:= FALSE;
		tyP0928MagConv.tyTopDC.tyBtnMagOut.bRtCompl				:= FALSE;
		tyP0928MagConv.tyTopDC.tyBtnStop.bRtCompl				:= FALSE;

		tyP0928MagConv.tyTopDC.tyBtnMagIn.bValue				:= FALSE;
		tyP0928MagConv.tyTopDC.tyBtnMagOut.bValue				:= FALSE;
		tyP0928MagConv.tyTopDC.tyBtnStop.bValue					:= TRUE;

		tyP0928MagConv.tyTopDC.tyBtnMagIn.bRtLk					:= FALSE;
		tyP0928MagConv.tyTopDC.tyBtnMagOut.bRtLk				:= FALSE;
		tyP0928MagConv.tyTopDC.tyBtnStop.bRtLk					:= TRUE;

		tyP0928MagConv.tyTopDC.tyBtnMagIn.uiMaskRtStat.0		:= TRUE;
		tyP0928MagConv.tyTopDC.tyBtnMagOut.uiMaskRtStat.0		:= TRUE;
		tyP0928MagConv.tyCom.tyBtnSwitch.uiMaskRtStat.0			:= TRUE;

		//Magazine Clamper
		//FB
		//Top
		tyP0928MagConv.tyTopFB.tyBtnEntStprExt.bRtCompl			:= FALSE;
		tyP0928MagConv.tyTopFB.tyBtnEntStprRet.bRtCompl			:= FALSE;

		tyP0928MagConv.tyTopFB.tyBtnEntStprExt.bValue				:= FALSE;
		tyP0928MagConv.tyTopFB.tyBtnEntStprRet.bValue			:= FALSE;

		//Remote
		tyP0928MagConv.tyTopFB.tyBtnMidStprExt.bRtCompl			:= FALSE;
		tyP0928MagConv.tyTopFB.tyBtnMidStprRet.bRtCompl		:= FALSE;

		tyP0928MagConv.tyTopFB.tyBtnMidStprExt.bValue			:= FALSE;
		tyP0928MagConv.tyTopFB.tyBtnMidStprRet.bValue			:= FALSE;

		//Top
		tyP0928MagConv.tyTopFB.tyBtnExtStprExt.bRtCompl			:= FALSE;
		tyP0928MagConv.tyTopFB.tyBtnExtStprRet.bRtCompl		:= FALSE;

		tyP0928MagConv.tyTopFB.tyBtnExtStprExt.bValue			:= FALSE;
		tyP0928MagConv.tyTopFB.tyBtnExtStprRet.bValue			:= FALSE;

		tyP0928MagConv.tyTopFB.tyBtnEntStprExt.uiMaskRtStat.0		:= TRUE;
		tyP0928MagConv.tyTopFB.tyBtnEntStprRet.uiMaskRtStat.0	:= TRUE;
		tyP0928MagConv.tyTopFB.tyBtnMidStprExt.uiMaskRtStat.0	:= TRUE;
		tyP0928MagConv.tyTopFB.tyBtnMidStprRet.uiMaskRtStat.0	:= TRUE;
		tyP0928MagConv.tyTopFB.tyBtnExtStprExt.uiMaskRtStat.0		:= TRUE;
		tyP0928MagConv.tyTopFB.tyBtnExtStprRet.uiMaskRtStat.0		:= TRUE;

		tyP0928MagConv.tyCom.tyBtnSwitch.uiMaskRtStat.0		:= TRUE;

		//Direct
		//Fixed
		tyP0928MagConv.tyTopDC.tyBtnEntStprExt.bRtCompl			:= FALSE;
		tyP0928MagConv.tyTopDC.tyBtnEntStprRet.bRtCompl			:= FALSE;

		tyP0928MagConv.tyTopDC.tyBtnEntStprExt.bValue				:= FALSE;
		tyP0928MagConv.tyTopDC.tyBtnEntStprRet.bValue			:= FALSE;

		//Remote
		tyP0928MagConv.tyTopDC.tyBtnMidStprExt.bRtCompl			:= FALSE;
		tyP0928MagConv.tyTopDC.tyBtnMidStprRet.bRtCompl		:= FALSE;

		tyP0928MagConv.tyTopDC.tyBtnMidStprExt.bValue			:= FALSE;
		tyP0928MagConv.tyTopDC.tyBtnMidStprRet.bValue			:= FALSE;

		//Top
		tyP0928MagConv.tyTopDC.tyBtnExtStprExt.bRtCompl				:= FALSE;
		tyP0928MagConv.tyTopDC.tyBtnExtStprRet.bRtCompl			:= FALSE;

		tyP0928MagConv.tyTopDC.tyBtnExtStprExt.bValue				:= FALSE;
		tyP0928MagConv.tyTopDC.tyBtnExtStprRet.bValue				:= FALSE;

		tyP0928MagConv.tyTopDC.tyBtnEntStprExt.uiMaskRtStat.0		:= TRUE;
		tyP0928MagConv.tyTopDC.tyBtnEntStprRet.uiMaskRtStat.0	:= TRUE;
		tyP0928MagConv.tyTopDC.tyBtnMidStprExt.uiMaskRtStat.0	:= TRUE;
		tyP0928MagConv.tyTopDC.tyBtnMidStprRet.uiMaskRtStat.0	:= TRUE;
		tyP0928MagConv.tyTopDC.tyBtnExtStprExt.uiMaskRtStat.0		:= TRUE;
		tyP0928MagConv.tyTopDC.tyBtnExtStprRet.uiMaskRtStat.0		:= TRUE;

		tyP0928MagConv.tyCom.tyBtnSwitch.uiMaskRtStat.0		:= TRUE;

	END_IF

END_ACTION
```

#### Act_OptP0928RstMnlBtm.st
```iecst
ACTION Act_OptP0928RstMnlBtm:

	IF EDGEPOS((bManualMod = FALSE) OR (p_eOutMagConvStatus = Error)) THEN

		eOutMagConvAct	:= MagConvActIdle;
		//Magazine Conveyor
		//FB
		tyP0928MagConv.tyBtmFB.tyBtnEnt.bRtCompl				:= FALSE;
		tyP0928MagConv.tyBtmFB.tyBtnExit.bRtCompl				:= FALSE;
		tyP0928MagConv.tyBtmFB.tyBtnStop.bRtCompl				:= FALSE;

		tyP0928MagConv.tyBtmFB.tyBtnEnt.bValue				:= FALSE;
		tyP0928MagConv.tyBtmFB.tyBtnExit.bValue				:= FALSE;
		tyP0928MagConv.tyBtmFB.tyBtnStop.bValue				:= TRUE;

		tyP0928MagConv.tyBtmFB.tyBtnEnt.bRtLk				:= FALSE;
		tyP0928MagConv.tyBtmFB.tyBtnExit.bRtLk				:= FALSE;
		tyP0928MagConv.tyBtmFB.tyBtnStop.bRtLk				:= TRUE;

		tyP0928MagConv.tyBtmFB.tyBtnEnt.uiMaskRtStat.0		:= TRUE;
		tyP0928MagConv.tyBtmFB.tyBtnExit.uiMaskRtStat.0		:= TRUE;
		tyP0928MagConv.tyCom.tyBtnSwitch.uiMaskRtStat.0		:= TRUE;

		//Direct
		tyP0928MagConv.tyBtmDC.tyBtnMagIn.bRtCompl				:= FALSE;
		tyP0928MagConv.tyBtmDC.tyBtnMagOut.bRtCompl				:= FALSE;
		tyP0928MagConv.tyBtmDC.tyBtnStop.bRtCompl				:= FALSE;

		tyP0928MagConv.tyBtmDC.tyBtnMagIn.bValue				:= FALSE;
		tyP0928MagConv.tyBtmDC.tyBtnMagOut.bValue				:= FALSE;
		tyP0928MagConv.tyBtmDC.tyBtnStop.bValue					:= TRUE;

		tyP0928MagConv.tyBtmDC.tyBtnMagIn.bRtLk					:= FALSE;
		tyP0928MagConv.tyBtmDC.tyBtnMagOut.bRtLk				:= FALSE;
		tyP0928MagConv.tyBtmDC.tyBtnStop.bRtLk					:= TRUE;

		tyP0928MagConv.tyBtmDC.tyBtnMagIn.uiMaskRtStat.0		:= TRUE;
		tyP0928MagConv.tyBtmDC.tyBtnMagOut.uiMaskRtStat.0		:= TRUE;
		tyP0928MagConv.tyCom.tyBtnSwitch.uiMaskRtStat.0			:= TRUE;

		//Magazine Clamper
		//FB
		//Remote
		tyP0928MagConv.tyBtmFB.tyBtnMidStprExt.bRtCompl			:= FALSE;
		tyP0928MagConv.tyBtmFB.tyBtnMidStprRet.bRtCompl		:= FALSE;

		tyP0928MagConv.tyBtmFB.tyBtnMidStprExt.bValue			:= FALSE;
		tyP0928MagConv.tyBtmFB.tyBtnMidStprRet.bValue			:= FALSE;

		//Top
		tyP0928MagConv.tyBtmFB.tyBtnExtStprExt.bRtCompl			:= FALSE;
		tyP0928MagConv.tyBtmFB.tyBtnExtStprRet.bRtCompl		:= FALSE;

		tyP0928MagConv.tyBtmFB.tyBtnExtStprExt.bValue			:= FALSE;
		tyP0928MagConv.tyBtmFB.tyBtnExtStprRet.bValue			:= FALSE;

		tyP0928MagConv.tyBtmFB.tyBtnMidStprExt.uiMaskRtStat.0	:= TRUE;
		tyP0928MagConv.tyBtmFB.tyBtnMidStprRet.uiMaskRtStat.0	:= TRUE;
		tyP0928MagConv.tyBtmFB.tyBtnExtStprExt.uiMaskRtStat.0		:= TRUE;
		tyP0928MagConv.tyBtmFB.tyBtnExtStprRet.uiMaskRtStat.0		:= TRUE;

		tyP0928MagConv.tyCom.tyBtnSwitch.uiMaskRtStat.0		:= TRUE;

		//Direct
		//Fixed

		//Remote
		tyP0928MagConv.tyBtmDC.tyBtnMidStprExt.bRtCompl			:= FALSE;
		tyP0928MagConv.tyBtmDC.tyBtnMidStprRet.bRtCompl		:= FALSE;

		tyP0928MagConv.tyBtmDC.tyBtnMidStprExt.bValue			:= FALSE;
		tyP0928MagConv.tyBtmDC.tyBtnMidStprRet.bValue			:= FALSE;

		//Top
		tyP0928MagConv.tyBtmDC.tyBtnExtStprExt.bRtCompl				:= FALSE;
		tyP0928MagConv.tyBtmDC.tyBtnExtStprRet.bRtCompl			:= FALSE;

		tyP0928MagConv.tyBtmDC.tyBtnExtStprExt.bValue				:= FALSE;
		tyP0928MagConv.tyBtmDC.tyBtnExtStprRet.bValue				:= FALSE;

		tyP0928MagConv.tyBtmDC.tyBtnMidStprExt.uiMaskRtStat.0	:= TRUE;
		tyP0928MagConv.tyBtmDC.tyBtnMidStprRet.uiMaskRtStat.0	:= TRUE;
		tyP0928MagConv.tyBtmDC.tyBtnExtStprExt.uiMaskRtStat.0		:= TRUE;
		tyP0928MagConv.tyBtmDC.tyBtnExtStprRet.uiMaskRtStat.0		:= TRUE;

		tyP0928MagConv.tyCom.tyBtnSwitch.uiMaskRtStat.0		:= TRUE;

	END_IF

END_ACTION
```

#### Act_EntP0929Disp.st
```iecst
ACTION Act_EntP0929Disp:

	//Access Address
	p_tyC0002FullMask ACCESS ADR(tyP0929MagConv2.tyFullMaskHide);

	//p_tyC0004Navi ACCESS ADR(tyP0929MagConv2.tyNaviBack);

	p_tyC0004Navi ACCESS ADR(tyP0929MagConv2.tyNavi2Lyr);

	p_tyC0005Main ACCESS ADR(tyCommon.tyMain);

	p_tyC0007Notif ACCESS ADR(tyCommon.tyNotif);

	p_tyC0008MsgBox ACCESS ADR(tyP0929MagConv2.tyMsgBoxHide);

	p_tyC0009Info ACCESS ADR(tyCommon.tyInfo);

	p_tyP0929MagConv2Com ACCESS ADR(tyP0929MagConv2.tyCom);
	p_tyP0929MagConv2TopDC ACCESS ADR(tyP0929MagConv2.tyTopDC);
	p_tyP0929MagConv2TopFB ACCESS ADR(tyP0929MagConv2.tyTopFB);
	p_tyP0929MagConv2BtmDC ACCESS ADR(tyP0929MagConv2.tyBtmDC);
	p_tyP0929MagConv2BtmFB ACCESS ADR(tyP0929MagConv2.tyBtmFB);

	IF tyP0929MagConv2.tyCom.tyBtnSwitch.bValue AND tyP0929MagConv2.tyTopFB.tyLyr.uiRtStat = FALSE THEN
		fUIInRtStatHide(ADR(tyP0929MagConv2.tyTopFB.tyLyr.uiRtStat));
		fUIInRtStatOff(ADR(tyP0929MagConv2.tyTopDC.tyLyr.uiRtStat));
		fUIInRtStatHide(ADR(tyP0929MagConv2.tyBtmFB.tyLyr.uiRtStat));
		fUIInRtStatHide(ADR(tyP0929MagConv2.tyBtmDC.tyLyr.uiRtStat));

	ELSIF tyP0929MagConv2.tyCom.tyBtnSwitch.bValue AND tyP0929MagConv2.tyBtmFB.tyLyr.uiRtStat = FALSE THEN

		fUIInRtStatHide(ADR(tyP0929MagConv2.tyTopFB.tyLyr.uiRtStat));
		fUIInRtStatHide(ADR(tyP0929MagConv2.tyTopDC.tyLyr.uiRtStat));
		fUIInRtStatHide(ADR(tyP0929MagConv2.tyBtmFB.tyLyr.uiRtStat));
		fUIInRtStatOff(ADR(tyP0929MagConv2.tyBtmDC.tyLyr.uiRtStat));

	ELSIF tyP0929MagConv2.tyCom.tyBtnSwitch.bValue = FALSE AND tyP0929MagConv2.tyTopDC.tyLyr.uiRtStat = FALSE THEN
		fUIInRtStatOff(ADR(tyP0929MagConv2.tyTopFB.tyLyr.uiRtStat));
		fUIInRtStatHide(ADR(tyP0929MagConv2.tyTopDC.tyLyr.uiRtStat));
		fUIInRtStatHide(ADR(tyP0929MagConv2.tyBtmFB.tyLyr.uiRtStat));
		fUIInRtStatHide(ADR(tyP0929MagConv2.tyBtmDC.tyLyr.uiRtStat));

	ELSIF tyP0929MagConv2.tyCom.tyBtnSwitch.bValue = FALSE AND tyP0929MagConv2.tyBtmDC.tyLyr.uiRtStat = FALSE THEN
		fUIInRtStatHide(ADR(tyP0929MagConv2.tyTopFB.tyLyr.uiRtStat));
		fUIInRtStatHide(ADR(tyP0929MagConv2.tyTopDC.tyLyr.uiRtStat));
		fUIInRtStatOff(ADR(tyP0929MagConv2.tyBtmFB.tyLyr.uiRtStat));
		fUIInRtStatHide(ADR(tyP0929MagConv2.tyBtmDC.tyLyr.uiRtStat));

	END_IF

END_ACTION
```

#### Act_OptP0929FullMask.st
```iecst
ACTION Act_OptP0929FullMask:

	IF eCurrPage = UIP0929MagConv2 THEN

		IF p_tyDI.bEStopSig = FALSE THEN
			p_tyC0002FullMask ACCESS ADR(tyP0929MagConv2.tyFullMaskEStop);

		ELSIF p_tyDI.bCoverSWSig = FALSE THEN
			p_tyC0002FullMask ACCESS ADR(tyP0929MagConv2.tyFullMaskCWSig);

		ELSIF p_tyDI.bSafetyRlySig = FALSE THEN
			p_tyC0002FullMask ACCESS ADR(tyP0929MagConv2.tyFullMaskSafetyRly);

		ELSE
			p_tyC0002FullMask ACCESS ADR(tyP0929MagConv2.tyFullMaskHide);

		END_IF

	END_IF

END_ACTION
```

#### Act_OptP0929Navi.st
```iecst
ACTION Act_OptP0929Navi:

	IF tyP0929MagConv2.tyNavi2Lyr.tyBtnBack.bRtCompl = TRUE THEN
		tyP0929MagConv2.tyNavi2Lyr.tyBtnBack.bRtCompl	:= FALSE;
		tyP0929MagConv2.tyNavi2Lyr.tyBtnBack.bValue		:= FALSE;

		eChgPage	:= UIP0920MtrNPneuCtrl;
	END_IF

	IF p_tyNtParamCurr.bProjMagConvLane1Prep THEN

		IF (tyP0929MagConv2.tyNavi2Lyr.tyBtnLeft.bRtCompl OR tyP0929MagConv2.tyNavi2Lyr.tyBtnRgt.bRtCompl)
			AND tyP0929MagConv2.tyNavi2Lyr.tyBitmapPageDisp.usiValueIdx = 1 THEN
			tyP0929MagConv2.tyNavi2Lyr.tyBitmapPageDisp.usiValueIdx := 2;

			tyP0929MagConv2.tyNavi2Lyr.tyBtnLeft.bRtCompl	:= FALSE;
			tyP0929MagConv2.tyNavi2Lyr.tyBtnLeft.bValue		:= FALSE;
			tyP0929MagConv2.tyNavi2Lyr.tyBtnRgt.bRtCompl		:= FALSE;
			tyP0929MagConv2.tyNavi2Lyr.tyBtnRgt.bValue		:= FALSE;

			IF tyP0929MagConv2.tyCom.tyBtnSwitch.bValue = FALSE THEN
				//Layer (Bottom)
				tyP0929MagConv2.tyTopFB.tyLyr.uiRtStat 	:= TRUE;
				tyP0929MagConv2.tyTopDC.tyLyr.uiRtStat	:= TRUE;

				tyP0929MagConv2.tyBtmFB.tyLyr.uiRtStat 	:= FALSE;
				tyP0929MagConv2.tyBtmDC.tyLyr.uiRtStat	:= TRUE;
			ELSE //Direct ctrl
				tyP0929MagConv2.tyTopFB.tyLyr.uiRtStat 	:= TRUE;
				tyP0929MagConv2.tyTopDC.tyLyr.uiRtStat	:= TRUE;

				tyP0929MagConv2.tyBtmFB.tyLyr.uiRtStat 	:= TRUE;
				tyP0929MagConv2.tyBtmDC.tyLyr.uiRtStat	:= FALSE;
			END_IF
		ELSIF (tyP0929MagConv2.tyNavi2Lyr.tyBtnLeft.bRtCompl OR tyP0929MagConv2.tyNavi2Lyr.tyBtnRgt.bRtCompl)
			AND tyP0929MagConv2.tyNavi2Lyr.tyBitmapPageDisp.usiValueIdx = 2 THEN
			tyP0929MagConv2.tyNavi2Lyr.tyBitmapPageDisp.usiValueIdx := 1;

			tyP0929MagConv2.tyNavi2Lyr.tyBtnLeft.bRtCompl	:= FALSE;
			tyP0929MagConv2.tyNavi2Lyr.tyBtnLeft.bValue		:= FALSE;
			tyP0929MagConv2.tyNavi2Lyr.tyBtnRgt.bRtCompl		:= FALSE;
			tyP0929MagConv2.tyNavi2Lyr.tyBtnRgt.bValue		:= FALSE;

			IF tyP0929MagConv2.tyCom.tyBtnSwitch.bValue = FALSE THEN
				//Layer (Top)
				tyP0929MagConv2.tyTopFB.tyLyr.uiRtStat 	:= FALSE;
				tyP0929MagConv2.tyTopDC.tyLyr.uiRtStat	:= TRUE;

				tyP0929MagConv2.tyBtmFB.tyLyr.uiRtStat 	:= TRUE;
				tyP0929MagConv2.tyBtmDC.tyLyr.uiRtStat	:= TRUE;
			ELSE //direct ctrl
				tyP0929MagConv2.tyTopFB.tyLyr.uiRtStat 	:= TRUE;
				tyP0929MagConv2.tyTopDC.tyLyr.uiRtStat	:= FALSE;

				tyP0929MagConv2.tyBtmFB.tyLyr.uiRtStat 	:= TRUE;
				tyP0929MagConv2.tyBtmDC.tyLyr.uiRtStat	:= TRUE;
			END_IF
		END_IF

	END_IF
	tyP0929MagConv2.tyCom.tyBtnLane.uiRtStat := NOT(p_tyNtParamCurr.bProjMagConvLane2Prep);

	IF tyP0929MagConv2.tyCom.tyBtnLane.bRtCompl THEN
		tyP0929MagConv2.tyCom.tyBtnLane.bRtCompl := FALSE;
		tyP0929MagConv2.tyCom.tyBtnLane.bValue := FALSE;
		eChgPage			:= UIP0928MagConv;
	END_IF

END_ACTION
```

#### Act_OptP0929MagConv2ChgLyr.st
```iecst
ACTION Act_OptP0929MagConv2ChgLyr:

	IF tyP0929MagConv2.tyNavi2Lyr.tyBitmapPageDisp.usiValueIdx = 1 THEN //Top layer

		IF tyP0929MagConv2.tyCom.tyBtnSwitch.bRtCompl THEN
			tyP0929MagConv2.tyCom.tyBtnSwitch.bRtCompl	:= FALSE;

			IF tyP0929MagConv2.tyCom.tyBtnSwitch.bValue = TRUE THEN
				fUIInRtStatOff(ADR(tyP0929MagConv2.tyTopDC.tyLyr.uiRtStat));
				fUIInRtStatHide(ADR(tyP0929MagConv2.tyTopFB.tyLyr.uiRtStat));
			ELSE
				fUIInRtStatHide(ADR(tyP0929MagConv2.tyTopDC.tyLyr.uiRtStat));
				fUIInRtStatOff(ADR(tyP0929MagConv2.tyTopFB.tyLyr.uiRtStat));
			END_IF

		END_IF
	ELSIF tyP0929MagConv2.tyNavi2Lyr.tyBitmapPageDisp.usiValueIdx = 2 THEN ///Btm layer
		IF tyP0929MagConv2.tyCom.tyBtnSwitch.bRtCompl THEN
			tyP0929MagConv2.tyCom.tyBtnSwitch.bRtCompl	:= FALSE;

			IF tyP0929MagConv2.tyCom.tyBtnSwitch.bValue = TRUE THEN
				fUIInRtStatOff(ADR(tyP0929MagConv2.tyBtmDC.tyLyr.uiRtStat));
				fUIInRtStatHide(ADR(tyP0929MagConv2.tyBtmFB.tyLyr.uiRtStat));
			ELSE
				fUIInRtStatHide(ADR(tyP0929MagConv2.tyBtmDC.tyLyr.uiRtStat));
				fUIInRtStatOff(ADR(tyP0929MagConv2.tyBtmFB.tyLyr.uiRtStat));
			END_IF

		END_IF
	END_IF

END_ACTION
```

#### Act_OptP0929MagConv2Sen.st
```iecst
ACTION Act_OptP0929MagConv2Sen:
	// connect sensors to inputs
	tyP0929MagConv2.tyCom.tyBtnTopEntSen.bValue			:= p_tyDI.bInMagConv2EntSen;
	tyP0929MagConv2.tyCom.tyBtnTopMidSen.bValue			:= p_tyDI.bInMagConv2MidSen;
	tyP0929MagConv2.tyCom.tyBtnTopExtSen.bValue			:= p_tyDI.bInMagConv2ExtSen;
	tyP0929MagConv2.tyCom.tyBtnBtmEntSen.bValue			:= p_tyDI.bOutMagConv2EntSen;
	tyP0929MagConv2.tyCom.tyBtnBtmMidSen.bValue			:= p_tyDI.bOutMagConv2MidSen;
	tyP0929MagConv2.tyCom.tyBtnBtmExtSen.bValue			:= p_tyDI.bOutMagConv2ExtSen;

	//Machine Bitmap
	IF p_tyNtParamCurr.bProjMagConvLane2Prep THEN
		IF tyP0929MagConv2.tyNavi2Lyr.tyBitmapPageDisp.usiValueIdx = 1 THEN //Top layer
			tyP0929MagConv2.tyCom.tyBitmapMc.uiValueIdx := 0;
		ELSIF tyP0929MagConv2.tyNavi2Lyr.tyBitmapPageDisp.usiValueIdx = 2 THEN
			tyP0929MagConv2.tyCom.tyBitmapMc.uiValueIdx := 1;
		END_IF
	END_IF

END_ACTION
```

#### Act_OptP0929MagConv2TopFB.st
```iecst
ACTION Act_OptP0929MagConv2TopFB:

	//Magazine Conv2eyor
	IF tyP0929MagConv2.tyTopFB.tyBtnStop.bRtCompl = TRUE THEN
		eInMagConv2Act	:= MagConvActStop;

		IF p_eInMagConv2Stat = MagConvActStop AND p_eInMagConv2Status = Done THEN
			eInMagConv2Act	:= MagConvActIdle;

			tyP0929MagConv2.tyTopFB.tyBtnEnt.bRtCompl	:= FALSE;
			tyP0929MagConv2.tyTopFB.tyBtnEnt.bValue		:= FALSE;
			tyP0929MagConv2.tyTopFB.tyBtnEnt.bRtLk		:= FALSE;

			tyP0929MagConv2.tyTopFB.tyBtnExit.bRtCompl	:= FALSE;
			tyP0929MagConv2.tyTopFB.tyBtnExit.bValue	:= FALSE;
			tyP0929MagConv2.tyTopFB.tyBtnExit.bRtLk		:= FALSE;

			tyP0929MagConv2.tyTopFB.tyBtnStop.bRtCompl	:= FALSE;
			tyP0929MagConv2.tyTopFB.tyBtnStop.bValue	:= TRUE;
			tyP0929MagConv2.tyTopFB.tyBtnStop.bRtLk		:= TRUE;
		END_IF

	ELSIF tyP0929MagConv2.tyTopFB.tyBtnEnt.bRtCompl = TRUE THEN
		tyP0929MagConv2.tyTopFB.tyBtnEnt.bValue		:= TRUE;
		tyP0929MagConv2.tyTopFB.tyBtnEnt.bRtLk		:= TRUE;

		tyP0929MagConv2.tyTopFB.tyBtnStop.bValue	:= FALSE;
		tyP0929MagConv2.tyTopFB.tyBtnStop.bRtLk		:= FALSE;

		eInMagConv2Act	:= MagConvActEnt;

		IF p_eInMagConv2Stat = MagConvActEnt AND p_eInMagConv2Status = Done THEN
			eInMagConv2Act	:= MagConvActIdle;

			tyP0929MagConv2.tyTopFB.tyBtnEnt.bRtCompl	:= FALSE;

			tyP0929MagConv2.tyTopFB.tyBtnEnt.bValue	:= FALSE;
			tyP0929MagConv2.tyTopFB.tyBtnEnt.bRtLk		:= FALSE;

			tyP0929MagConv2.tyTopFB.tyBtnStop.bValue	:= TRUE;
			tyP0929MagConv2.tyTopFB.tyBtnStop.bRtLk	:= TRUE;
		END_IF

	ELSIF tyP0929MagConv2.tyTopFB.tyBtnExit.bRtCompl = TRUE THEN
		tyP0929MagConv2.tyTopFB.tyBtnExit.bValue	:= TRUE;
		tyP0929MagConv2.tyTopFB.tyBtnExit.bRtLk		:= TRUE;

		tyP0929MagConv2.tyTopFB.tyBtnStop.bValue	:= FALSE;
		tyP0929MagConv2.tyTopFB.tyBtnStop.bRtLk		:= FALSE;

		eInMagConv2Act	:= MagConvActExit;

		IF p_eInMagConv2Stat = MagConvActExit AND p_eInMagConv2Status = Done THEN
			eInMagConv2Act	:= MagConvActIdle;

			tyP0929MagConv2.tyTopFB.tyBtnExit.bRtCompl:= FALSE;

			tyP0929MagConv2.tyTopFB.tyBtnExit.bValue	:= FALSE;
			tyP0929MagConv2.tyTopFB.tyBtnExit.bRtLk	:= FALSE;

			tyP0929MagConv2.tyTopFB.tyBtnStop.bValue	:= TRUE;
			tyP0929MagConv2.tyTopFB.tyBtnStop.bRtLk	:= TRUE;
		END_IF
	END_IF

	//Stopper
	IF tyP0929MagConv2.tyCom.tyBtnSwitch.bValue = FALSE THEN

		//Ent Stopper
		IF tyP0929MagConv2.tyTopFB.tyBtnEntStprExt.bRtCompl = TRUE THEN
			tyP0929MagConv2.tyTopFB.tyBtnEntStprExt.bRtCompl	:= FALSE;

			tyP0929MagConv2.tyTopFB.tyBtnEntStprExt.bValue	:= TRUE;
			tyP0929MagConv2.tyTopFB.tyBtnEntStprRet.bValue		:= FALSE;

		ELSIF tyP0929MagConv2.tyTopFB.tyBtnEntStprRet.bRtCompl = TRUE THEN
			tyP0929MagConv2.tyTopFB.tyBtnEntStprRet.bRtCompl	:= FALSE;

			tyP0929MagConv2.tyTopFB.tyBtnEntStprRet.bValue		:= TRUE;
			tyP0929MagConv2.tyTopFB.tyBtnEntStprExt.bValue	:= FALSE;

		END_IF

		//Mid stopper
		IF tyP0929MagConv2.tyTopFB.tyBtnMidStprExt.bRtCompl = TRUE THEN
			tyP0929MagConv2.tyTopFB.tyBtnMidStprExt.bRtCompl	:= FALSE;

			tyP0929MagConv2.tyTopFB.tyBtnMidStprExt.bValue	:= TRUE;
			tyP0929MagConv2.tyTopFB.tyBtnMidStprRet.bValue	:= FALSE;

		ELSIF tyP0929MagConv2.tyTopFB.tyBtnMidStprRet.bRtCompl = TRUE THEN
			tyP0929MagConv2.tyTopFB.tyBtnMidStprRet.bRtCompl	:= FALSE;

			tyP0929MagConv2.tyTopFB.tyBtnMidStprRet.bValue	:= TRUE;
			tyP0929MagConv2.tyTopFB.tyBtnMidStprExt.bValue	:= FALSE;

		END_IF

		//Ext Stopper
		IF tyP0929MagConv2.tyTopFB.tyBtnExtStprExt.bRtCompl = TRUE THEN
			tyP0929MagConv2.tyTopFB.tyBtnExtStprExt.bRtCompl	:= FALSE;

			tyP0929MagConv2.tyTopFB.tyBtnExtStprExt.bValue	:= TRUE;
			tyP0929MagConv2.tyTopFB.tyBtnExtStprRet.bValue	:= FALSE;

		ELSIF tyP0929MagConv2.tyTopFB.tyBtnExtStprRet.bRtCompl = TRUE THEN
			tyP0929MagConv2.tyTopFB.tyBtnExtStprRet.bRtCompl	:= FALSE;

			tyP0929MagConv2.tyTopFB.tyBtnExtStprRet.bValue	:= TRUE;
			tyP0929MagConv2.tyTopFB.tyBtnExtStprExt.bValue	:= FALSE;

		END_IF

		//Action------------
		IF tyP0929MagConv2.tyTopFB.tyBtnEntStprExt.bValue = TRUE THEN
			eStopper1Act2	:= PneuActExt;

			IF p_eStopper1Stat2 = PneuActExt AND p_eStopper1Status2 = Done THEN
				eStopper1Act2	:= PneuActIdle;
				tyP0929MagConv2.tyTopFB.tyBtnEntStprExt.bValue	:= FALSE;
			ELSIF p_eStopper1Status2 = Error THEN
				tyP0929MagConv2.tyTopFB.tyBtnEntStprExt.bValue	:= FALSE;
			END_IF

		ELSIF tyP0929MagConv2.tyTopFB.tyBtnEntStprRet.bValue = TRUE THEN
			eStopper1Act2	:= PneuActRet;

			IF p_eStopper1Stat2 = PneuActRet AND p_eStopper1Status2 = Done THEN
				eStopper1Act2	:= PneuActIdle;
				tyP0929MagConv2.tyTopFB.tyBtnEntStprRet.bValue := FALSE;
			ELSIF p_eStopper1Status2 = Error THEN
				tyP0929MagConv2.tyTopFB.tyBtnEntStprRet.bValue := FALSE;
			END_IF

		END_IF

		IF tyP0929MagConv2.tyTopFB.tyBtnMidStprExt.bValue = TRUE THEN
			eStopper2Act2	:= PneuActExt;

			IF p_eStopper2Stat2 = PneuActExt AND p_eStopper2Status2 = Done THEN
				eStopper2Act2	:= PneuActIdle;
				tyP0929MagConv2.tyTopFB.tyBtnMidStprExt.bValue	:= FALSE;
			ELSIF p_eStopper2Status2 = Error THEN
				tyP0929MagConv2.tyTopFB.tyBtnMidStprExt.bValue	:= FALSE;
			END_IF

		ELSIF tyP0929MagConv2.tyTopFB.tyBtnMidStprRet.bValue = TRUE THEN
			eStopper2Act2	:= PneuActRet;

			IF p_eStopper2Stat2 = PneuActRet AND p_eStopper2Status2 = Done THEN
				eStopper2Act2	:= PneuActIdle;
				tyP0929MagConv2.tyTopFB.tyBtnMidStprRet.bValue := FALSE;
			ELSIF p_eStopper2Status2 = Error THEN
				tyP0929MagConv2.tyTopFB.tyBtnMidStprRet.bValue := FALSE;
			END_IF

		END_IF

		IF tyP0929MagConv2.tyTopFB.tyBtnExtStprExt.bValue = TRUE THEN
			eStopper3Act2	:= PneuActExt;

			IF p_eStopper3Stat2 = PneuActExt AND p_eStopper3Status2 = Done THEN
				eStopper3Act2	:= PneuActIdle;
				tyP0929MagConv2.tyTopFB.tyBtnExtStprExt.bValue	:= FALSE;
			ELSIF p_eStopper3Status2 = Error THEN
				tyP0929MagConv2.tyTopFB.tyBtnExtStprExt.bValue	:= FALSE;
			END_IF

		ELSIF tyP0929MagConv2.tyTopFB.tyBtnExtStprRet.bValue = TRUE THEN
			eStopper3Act2	:= PneuActRet;

			IF p_eStopper3Stat2 = PneuActRet AND p_eStopper3Status2 = Done THEN
				eStopper3Act2	:= PneuActIdle;
				tyP0929MagConv2.tyTopFB.tyBtnExtStprRet.bValue := FALSE;
			ELSIF p_eStopper3Status2 = Error THEN
				tyP0929MagConv2.tyTopFB.tyBtnExtStprRet.bValue := FALSE;
			END_IF

		END_IF

		//Update Status
//		tyP0929MagConv2.tyDC.tyBtnFixedUnclamp.bValue	:= NOT p_bStopper1RetCtrl2;
//		tyP0929MagConv2.tyDC.tyBtnFixedClamp.bValue		:= p_bMagConv22Clp1ClprFixClampCtrl;
//		tyP0929MagConv2.tyDC.tyBtnRemoteUnclamp.bValue	:= NOT p_bMagConv22Clp1ClprRmtClampCtrl;
//		tyP0929MagConv2.tyDC.tyBtnRemoteClamp.bValue	:= p_bMagConv22Clp1ClprRmtClampCtrl;
//
//		tyP0929MagConv2.tyDC.tyBtnSelUnclamp.bRtCompl	:= FALSE;
//		tyP0929MagConv2.tyDC.tyBtnSelClamp.bRtCompl		:= FALSE;
//		tyP0929MagConv2.tyDC.tyBtnSelUnclamp.bValue	:= p_bSelClamp1RetCtrl;
//		tyP0929MagConv2.tyDC.tyBtnSelClamp.bValue	:= p_bSelClamp1ExtCtrl;
	END_IF

	//Mask
//	IF p_tyUsrMgmtCurrAccessRgt.bManualFBOnly THEN
//
//		fUIInRtStatOff(ADR(tyP0929MagConv2.tyCom.tyBtnSwitch.uiMaskRtStat));
//
//	ELSE
//
//		IF p_eInMagConv2Status = Error THEN
//
//			fUIInRtStatOff(ADR(tyP0929MagConv2.tyTopFB.tyBtnEnt.uiMaskRtStat));
//			fUIInRtStatOff(ADR(tyP0929MagConv2.tyTopFB.tyBtnExit.uiMaskRtStat));
//			fUIInRtStatOff(ADR(tyP0929MagConv2.tyTopFB.tyBtnEntStprExt.uiMaskRtStat));
//			fUIInRtStatOff(ADR(tyP0929MagConv2.tyTopFB.tyBtnEntStprRet.uiMaskRtStat));
//			fUIInRtStatOff(ADR(tyP0929MagConv2.tyTopFB.tyBtnMidStprExt.uiMaskRtStat));
//			fUIInRtStatOff(ADR(tyP0929MagConv2.tyTopFB.tyBtnMidStprRet.uiMaskRtStat));
//			fUIInRtStatOff(ADR(tyP0929MagConv2.tyTopFB.tyBtnExtStprExt.uiMaskRtStat));
//			fUIInRtStatOff(ADR(tyP0929MagConv2.tyTopFB.tyBtnExtStprRet.uiMaskRtStat));
//			fUIInRtStatHide(ADR(tyP0929MagConv2.tyCom.tyBtnSwitch.uiMaskRtStat));
//
//		ELSIF tyP0929MagConv2.tyTopFB.tyBtnEnt.bRtCompl = TRUE THEN
//
//			fUIInRtStatHide(ADR(tyP0929MagConv2.tyTopFB.tyBtnEnt.uiMaskRtStat));
//			fUIInRtStatOff(ADR(tyP0929MagConv2.tyTopFB.tyBtnExit.uiMaskRtStat));
//			fUIInRtStatOff(ADR(tyP0929MagConv2.tyTopFB.tyBtnFixedClamp.uiMaskRtStat));
//			fUIInRtStatOff(ADR(tyP0929MagConv2.tyTopFB.tyBtnFixedUnclamp.uiMaskRtStat));
//			fUIInRtStatOff(ADR(tyP0929MagConv2.tyTopFB.tyBtnRemoteClamp.uiMaskRtStat));
//			fUIInRtStatOff(ADR(tyP0929MagConv2.tyTopFB.tyBtnRemoteUnclamp.uiMaskRtStat));
//			fUIInRtStatOff(ADR(tyP0929MagConv2.tyTopFB.tyBtnSelClamp.uiMaskRtStat));
//			fUIInRtStatOff(ADR(tyP0929MagConv2.tyTopFB.tyBtnSelUnclamp.uiMaskRtStat));
//			fUIInRtStatOff(ADR(tyP0929MagConv2.tyCom.tyBtnSwitch.uiMaskRtStat));
//
//		ELSIF tyP0929MagConv2.tyTopFB.tyBtnExit.bRtCompl = TRUE THEN
//
//			fUIInRtStatOff(ADR(tyP0929MagConv2.tyTopFB.tyBtnEnt.uiMaskRtStat));
//			fUIInRtStatHide(ADR(tyP0929MagConv2.tyTopFB.tyBtnExit.uiMaskRtStat));
//			fUIInRtStatOff(ADR(tyP0929MagConv2.tyTopFB.tyBtnFixedClamp.uiMaskRtStat));
//			fUIInRtStatOff(ADR(tyP0929MagConv2.tyTopFB.tyBtnFixedUnclamp.uiMaskRtStat));
//			fUIInRtStatOff(ADR(tyP0929MagConv2.tyTopFB.tyBtnRemoteClamp.uiMaskRtStat));
//			fUIInRtStatOff(ADR(tyP0929MagConv2.tyTopFB.tyBtnRemoteUnclamp.uiMaskRtStat));
//			fUIInRtStatOff(ADR(tyP0929MagConv2.tyTopFB.tyBtnSelClamp.uiMaskRtStat));
//			fUIInRtStatOff(ADR(tyP0929MagConv2.tyTopFB.tyBtnSelUnclamp.uiMaskRtStat));
//			fUIInRtStatOff(ADR(tyP0929MagConv2.tyCom.tyBtnSwitch.uiMaskRtStat));
//
//		ELSIF tyP0929MagConv2.tyTopFB.tyBtnFixedClamp.bValue = TRUE OR tyP0929MagConv2.tyTopFB.tyBtnRemoteClamp.bValue = TRUE
//			OR tyP0929MagConv2.tyTopFB.tyBtnFixedUnclamp.bValue = TRUE OR tyP0929MagConv2.tyTopFB.tyBtnRemoteUnclamp.bValue = TRUE
//			OR tyP0929MagConv2.tyTopFB.tyBtnSelUnclamp.bValue = TRUE OR tyP0929MagConv2.tyTopFB.tyBtnSelClamp.bValue = TRUE
//			THEN
//
//			fUIInRtStatOff(ADR(tyP0929MagConv2.tyTopFB.tyBtnEnt.uiMaskRtStat));
//			fUIInRtStatOff(ADR(tyP0929MagConv2.tyTopFB.tyBtnExit.uiMaskRtStat));
//			fUIInRtStatHide(ADR(tyP0929MagConv2.tyTopFB.tyBtnFixedClamp.uiMaskRtStat));
//		fUIInRtStatHide(ADR(tyP0929MagConv2.tyTopFB.tyBtnFixedUnclamp.uiMaskRtStat));
//		fUIInRtStatHide(ADR(tyP0929MagConv2.tyTopFB.tyBtnRemoteClamp.uiMaskRtStat));
//		fUIInRtStatHide(ADR(tyP0929MagConv2.tyTopFB.tyBtnRemoteUnclamp.uiMaskRtStat));
//		fUIInRtStatHide(ADR(tyP0929MagConv2.tyTopFB.tyBtnSelClamp.uiMaskRtStat));
//		fUIInRtStatHide(ADR(tyP0929MagConv2.tyTopFB.tyBtnSelUnclamp.uiMaskRtStat));
//		fUIInRtStatOff(ADR(tyP0929MagConv2.tyCom.tyBtnSwitch.uiMaskRtStat));
//
//	ELSE
//
//		fUIInRtStatHide(ADR(tyP0929MagConv2.tyTopFB.tyBtnEnt.uiMaskRtStat));
//		fUIInRtStatHide(ADR(tyP0929MagConv2.tyTopFB.tyBtnExit.uiMaskRtStat));
//		fUIInRtStatHide(ADR(tyP0929MagConv2.tyTopFB.tyBtnFixedClamp.uiMaskRtStat));
//		fUIInRtStatHide(ADR(tyP0929MagConv2.tyTopFB.tyBtnFixedUnclamp.uiMaskRtStat));
//		fUIInRtStatHide(ADR(tyP0929MagConv2.tyTopFB.tyBtnRemoteClamp.uiMaskRtStat));
//		fUIInRtStatHide(ADR(tyP0929MagConv2.tyTopFB.tyBtnRemoteUnclamp.uiMaskRtStat));
//		fUIInRtStatHide(ADR(tyP0929MagConv2.tyTopFB.tyBtnSelClamp.uiMaskRtStat));
//		fUIInRtStatHide(ADR(tyP0929MagConv2.tyTopFB.tyBtnSelUnclamp.uiMaskRtStat));
//		fUIInRtStatHide(ADR(tyP0929MagConv2.tyCom.tyBtnSwitch.uiMaskRtStat));
//
//	END_IF
//END_IF

END_ACTION
```

#### Act_OptP0929MagConv2FBStat.st
```iecst
ACTION Act_OptP0929MagConv2FBStat:

	IF tyP0929MagConv2.tyTopFB.tyBtnEntStprExt.bValue OR tyP0929MagConv2.tyTopFB.tyBtnEntStprRet.bValue THEN
		tyP0929MagConv2.tyTopFB.tyStringStat.sValue	:= p_sStopper1StatTxt2;
	ELSIF tyP0929MagConv2.tyTopFB.tyBtnMidStprExt.bValue OR tyP0929MagConv2.tyTopFB.tyBtnMidStprRet.bValue THEN
		tyP0929MagConv2.tyTopFB.tyStringStat.sValue	:= p_sStopper2StatTxt2;
	ELSIF tyP0929MagConv2.tyTopFB.tyBtnExtStprExt.bValue OR tyP0929MagConv2.tyTopFB.tyBtnExtStprRet.bValue THEN
		tyP0929MagConv2.tyTopFB.tyStringStat.sValue	:= p_sStopper3StatTxt2;

	ELSIF tyP0929MagConv2.tyBtmFB.tyBtnMidStprExt.bValue OR tyP0929MagConv2.tyBtmFB.tyBtnMidStprRet.bValue THEN
		tyP0929MagConv2.tyBtmFB.tyStringStat.sValue	:= p_sStopper4StatTxt2;
	ELSIF tyP0929MagConv2.tyBtmFB.tyBtnExtStprExt.bValue OR tyP0929MagConv2.tyBtmFB.tyBtnExtStprRet.bValue THEN
		tyP0929MagConv2.tyBtmFB.tyStringStat.sValue	:= p_sStopper5StatTxt2;

	ELSIF tyP0929MagConv2.tyTopFB.tyBtnEnt.bValue OR tyP0929MagConv2.tyTopFB.tyBtnExit.bValue THEN
		tyP0929MagConv2.tyTopFB.tyStringStat.sValue	:= p_sInMagConv2StatTxt;
	ELSIF tyP0929MagConv2.tyBtmFB.tyBtnEnt.bValue OR tyP0929MagConv2.tyBtmFB.tyBtnExit.bValue THEN
		tyP0929MagConv2.tyBtmFB.tyStringStat.sValue	:= p_sOutMagConv2StatTxt;

	END_IF

END_ACTION
```

#### Act_OptP0929MagConv2BtmFB.st
```iecst
ACTION Act_OptP0929MagConv2BtmFB:

	//Magazine Conv2eyor
	IF tyP0929MagConv2.tyBtmFB.tyBtnStop.bRtCompl = TRUE THEN
		eOutMagConv2Act	:= MagConvActStop;

		IF p_eOutMagConv2Stat = MagConvActStop AND p_eOutMagConv2Status = Done THEN
			eOutMagConv2Act	:= MagConvActIdle;

			tyP0929MagConv2.tyBtmFB.tyBtnEnt.bRtCompl	:= FALSE;
			tyP0929MagConv2.tyBtmFB.tyBtnEnt.bValue		:= FALSE;
			tyP0929MagConv2.tyBtmFB.tyBtnEnt.bRtLk		:= FALSE;

			tyP0929MagConv2.tyBtmFB.tyBtnExit.bRtCompl	:= FALSE;
			tyP0929MagConv2.tyBtmFB.tyBtnExit.bValue		:= FALSE;
			tyP0929MagConv2.tyBtmFB.tyBtnExit.bRtLk		:= FALSE;

			tyP0929MagConv2.tyBtmFB.tyBtnStop.bRtCompl	:= FALSE;
			tyP0929MagConv2.tyBtmFB.tyBtnStop.bValue		:= TRUE;
			tyP0929MagConv2.tyBtmFB.tyBtnStop.bRtLk		:= TRUE;
		END_IF

	ELSIF tyP0929MagConv2.tyBtmFB.tyBtnEnt.bRtCompl = TRUE THEN
		tyP0929MagConv2.tyBtmFB.tyBtnEnt.bValue	:= TRUE;
		tyP0929MagConv2.tyBtmFB.tyBtnEnt.bRtLk		:= TRUE;

		tyP0929MagConv2.tyBtmFB.tyBtnStop.bValue	:= FALSE;
		tyP0929MagConv2.tyBtmFB.tyBtnStop.bRtLk	:= FALSE;

		eOutMagConv2Act	:= MagConvActEnt;

		IF p_eOutMagConv2Stat = MagConvActEnt AND p_eOutMagConv2Status = Done THEN
			eOutMagConv2Act	:= MagConvActIdle;

			tyP0929MagConv2.tyBtmFB.tyBtnEnt.bRtCompl	:= FALSE;

			tyP0929MagConv2.tyBtmFB.tyBtnEnt.bValue	:= FALSE;
			tyP0929MagConv2.tyBtmFB.tyBtnEnt.bRtLk		:= FALSE;

			tyP0929MagConv2.tyBtmFB.tyBtnStop.bValue	:= TRUE;
			tyP0929MagConv2.tyBtmFB.tyBtnStop.bRtLk	:= TRUE;
		END_IF

	ELSIF tyP0929MagConv2.tyBtmFB.tyBtnExit.bRtCompl = TRUE THEN
		tyP0929MagConv2.tyBtmFB.tyBtnExit.bValue	:= TRUE;
		tyP0929MagConv2.tyBtmFB.tyBtnExit.bRtLk	:= TRUE;

		tyP0929MagConv2.tyBtmFB.tyBtnStop.bValue	:= FALSE;
		tyP0929MagConv2.tyBtmFB.tyBtnStop.bRtLk	:= FALSE;

		eOutMagConv2Act	:= MagConvActExit;

		IF p_eOutMagConv2Stat = MagConvActExit AND p_eOutMagConv2Status = Done THEN
			eOutMagConv2Act	:= MagConvActIdle;

			tyP0929MagConv2.tyBtmFB.tyBtnExit.bRtCompl:= FALSE;

			tyP0929MagConv2.tyBtmFB.tyBtnExit.bValue	:= FALSE;
			tyP0929MagConv2.tyBtmFB.tyBtnExit.bRtLk	:= FALSE;

			tyP0929MagConv2.tyBtmFB.tyBtnStop.bValue	:= TRUE;
			tyP0929MagConv2.tyBtmFB.tyBtnStop.bRtLk	:= TRUE;
		END_IF
	END_IF

	//Stopper
	IF tyP0929MagConv2.tyCom.tyBtnSwitch.bValue = FALSE THEN

		//Mid stopper
		IF tyP0929MagConv2.tyBtmFB.tyBtnMidStprExt.bRtCompl = TRUE THEN
			tyP0929MagConv2.tyBtmFB.tyBtnMidStprExt.bRtCompl	:= FALSE;

			tyP0929MagConv2.tyBtmFB.tyBtnMidStprExt.bValue	:= TRUE;
			tyP0929MagConv2.tyBtmFB.tyBtnMidStprRet.bValue	:= FALSE;

		ELSIF tyP0929MagConv2.tyBtmFB.tyBtnMidStprRet.bRtCompl = TRUE THEN
			tyP0929MagConv2.tyBtmFB.tyBtnMidStprRet.bRtCompl	:= FALSE;

			tyP0929MagConv2.tyBtmFB.tyBtnMidStprRet.bValue	:= TRUE;
			tyP0929MagConv2.tyBtmFB.tyBtnMidStprExt.bValue	:= FALSE;

		END_IF

		//Ext Stopper
		IF tyP0929MagConv2.tyBtmFB.tyBtnExtStprExt.bRtCompl = TRUE THEN
			tyP0929MagConv2.tyBtmFB.tyBtnExtStprExt.bRtCompl	:= FALSE;

			tyP0929MagConv2.tyBtmFB.tyBtnExtStprExt.bValue	:= TRUE;
			tyP0929MagConv2.tyBtmFB.tyBtnExtStprRet.bValue	:= FALSE;

		ELSIF tyP0929MagConv2.tyBtmFB.tyBtnExtStprRet.bRtCompl = TRUE THEN
			tyP0929MagConv2.tyBtmFB.tyBtnExtStprRet.bRtCompl	:= FALSE;

			tyP0929MagConv2.tyBtmFB.tyBtnExtStprRet.bValue	:= TRUE;
			tyP0929MagConv2.tyBtmFB.tyBtnExtStprExt.bValue	:= FALSE;

		END_IF

		//Action------------

		IF tyP0929MagConv2.tyBtmFB.tyBtnMidStprExt.bValue = TRUE THEN
				eStopper4Act2	:= PneuActExt;

				IF p_eStopper4Stat = PneuActExt AND p_eStopper4Status = Done THEN
					eStopper4Act2	:= PneuActIdle;
					tyP0929MagConv2.tyBtmFB.tyBtnMidStprExt.bValue	:= FALSE;
				ELSIF p_eStopper4Status = Error THEN
					tyP0929MagConv2.tyBtmFB.tyBtnMidStprExt.bValue	:= FALSE;
				END_IF

		ELSIF tyP0929MagConv2.tyBtmFB.tyBtnMidStprRet.bValue = TRUE THEN
			eStopper4Act2	:= PneuActRet;

			IF p_eStopper4Stat = PneuActRet AND p_eStopper4Status = Done THEN
				eStopper4Act2	:= PneuActIdle;
				tyP0929MagConv2.tyBtmFB.tyBtnMidStprRet.bValue := FALSE;
			ELSIF p_eStopper4Status = Error THEN
				tyP0929MagConv2.tyBtmFB.tyBtnMidStprRet.bValue := FALSE;
			END_IF

		END_IF

		IF tyP0929MagConv2.tyBtmFB.tyBtnExtStprExt.bValue = TRUE THEN
			eStopper5Act2	:= PneuActExt;

			IF p_eStopper5Stat = PneuActExt AND p_eStopper5Status = Done THEN
				eStopper5Act2	:= PneuActIdle;
				tyP0929MagConv2.tyBtmFB.tyBtnExtStprExt.bValue	:= FALSE;
			ELSIF p_eStopper5Status = Error THEN
				tyP0929MagConv2.tyBtmFB.tyBtnExtStprExt.bValue	:= FALSE;
			END_IF

		ELSIF tyP0929MagConv2.tyBtmFB.tyBtnExtStprRet.bValue = TRUE THEN
			eStopper5Act2	:= PneuActRet;

			IF p_eStopper5Stat = PneuActRet AND p_eStopper5Status = Done THEN
				eStopper5Act2	:= PneuActIdle;
				tyP0929MagConv2.tyBtmFB.tyBtnExtStprRet.bValue := FALSE;
			ELSIF p_eStopper5Status = Error THEN
				tyP0929MagConv2.tyBtmFB.tyBtnExtStprRet.bValue := FALSE;
			END_IF

		END_IF

		//Update Status
//		tyP0930MagConv2Btm1.tyDC.tyBtnFixedUnclamp.bValue	:= NOT p_bMagConv2Btm2Clp1ClprFixClampCtrl;
//		tyP0930MagConv2Btm1.tyDC.tyBtnFixedClamp.bValue		:= p_bMagConv2Btm2Clp1ClprFixClampCtrl;
//		tyP0930MagConv2Btm1.tyDC.tyBtnRemoteUnclamp.bValue	:= NOT p_bMagConv2Btm2Clp1ClprRmtClampCtrl;
//		tyP0930MagConv2Btm1.tyDC.tyBtnRemoteClamp.bValue	:= p_bMagConv2Btm2Clp1ClprRmtClampCtrl;
//
//		tyP0930MagConv2Btm1.tyDC.tyBtnSelUnclamp.bRtCompl	:= FALSE;
//		tyP0930MagConv2Btm1.tyDC.tyBtnSelClamp.bRtCompl		:= FALSE;
//		tyP0930MagConv2Btm1.tyDC.tyBtnSelUnclamp.bValue	:= p_bSelClamp1RetCtrl;
//		tyP0930MagConv2Btm1.tyDC.tyBtnSelClamp.bValue	:= p_bSelClamp1ExtCtrl;
	END_IF

	//Mask
//	IF p_tyUsrMgmtCurrAccessRgt.bManualFBOnly THEN
//
//		fUIInRtStatOff(ADR(tyP0930MagConv2Btm1.tyCom.tyBtnSwitch.uiMaskRtStat));
//
//	ELSE
//
//	IF p_eMagConv2Btm2Clp1Status = Error THEN
//
//		fUIInRtStatOff(ADR(tyP0930MagConv2Btm1.tyFB.tyBtnEnt.uiMaskRtStat));
//		fUIInRtStatOff(ADR(tyP0930MagConv2Btm1.tyFB.tyBtnExit.uiMaskRtStat));
//		fUIInRtStatOff(ADR(tyP0930MagConv2Btm1.tyFB.tyBtnFixedClamp.uiMaskRtStat));
//		fUIInRtStatOff(ADR(tyP0930MagConv2Btm1.tyFB.tyBtnFixedUnclamp.uiMaskRtStat));
//		fUIInRtStatOff(ADR(tyP0930MagConv2Btm1.tyFB.tyBtnRemoteClamp.uiMaskRtStat));
//		fUIInRtStatOff(ADR(tyP0930MagConv2Btm1.tyFB.tyBtnRemoteUnclamp.uiMaskRtStat));
//		fUIInRtStatOff(ADR(tyP0930MagConv2Btm1.tyFB.tyBtnSelClamp.uiMaskRtStat));
//		fUIInRtStatOff(ADR(tyP0930MagConv2Btm1.tyFB.tyBtnSelUnclamp.uiMaskRtStat));
//		fUIInRtStatHide(ADR(tyP0930MagConv2Btm1.tyCom.tyBtnSwitch.uiMaskRtStat));
//
//	ELSIF tyP0930MagConv2Btm1.tyFB.tyBtnEnt.bRtCompl = TRUE THEN
//
//		fUIInRtStatHide(ADR(tyP0930MagConv2Btm1.tyFB.tyBtnEnt.uiMaskRtStat));
//		fUIInRtStatOff(ADR(tyP0930MagConv2Btm1.tyFB.tyBtnExit.uiMaskRtStat));
//		fUIInRtStatOff(ADR(tyP0930MagConv2Btm1.tyFB.tyBtnFixedClamp.uiMaskRtStat));
//		fUIInRtStatOff(ADR(tyP0930MagConv2Btm1.tyFB.tyBtnFixedUnclamp.uiMaskRtStat));
//		fUIInRtStatOff(ADR(tyP0930MagConv2Btm1.tyFB.tyBtnRemoteClamp.uiMaskRtStat));
//		fUIInRtStatOff(ADR(tyP0930MagConv2Btm1.tyFB.tyBtnRemoteUnclamp.uiMaskRtStat));
//		fUIInRtStatOff(ADR(tyP0930MagConv2Btm1.tyFB.tyBtnSelClamp.uiMaskRtStat));
//		fUIInRtStatOff(ADR(tyP0930MagConv2Btm1.tyFB.tyBtnSelUnclamp.uiMaskRtStat));
//		fUIInRtStatOff(ADR(tyP0930MagConv2Btm1.tyCom.tyBtnSwitch.uiMaskRtStat));
//
//	ELSIF tyP0930MagConv2Btm1.tyFB.tyBtnExit.bRtCompl = TRUE THEN
//
//			fUIInRtStatOff(ADR(tyP0930MagConv2Btm1.tyFB.tyBtnEnt.uiMaskRtStat));
//		fUIInRtStatHide(ADR(tyP0930MagConv2Btm1.tyFB.tyBtnExit.uiMaskRtStat));
//		fUIInRtStatOff(ADR(tyP0930MagConv2Btm1.tyFB.tyBtnFixedClamp.uiMaskRtStat));
//		fUIInRtStatOff(ADR(tyP0930MagConv2Btm1.tyFB.tyBtnFixedUnclamp.uiMaskRtStat));
//		fUIInRtStatOff(ADR(tyP0930MagConv2Btm1.tyFB.tyBtnRemoteClamp.uiMaskRtStat));
//		fUIInRtStatOff(ADR(tyP0930MagConv2Btm1.tyFB.tyBtnRemoteUnclamp.uiMaskRtStat));
//		fUIInRtStatOff(ADR(tyP0930MagConv2Btm1.tyFB.tyBtnSelClamp.uiMaskRtStat));
//		fUIInRtStatOff(ADR(tyP0930MagConv2Btm1.tyFB.tyBtnSelUnclamp.uiMaskRtStat));
//		fUIInRtStatOff(ADR(tyP0930MagConv2Btm1.tyCom.tyBtnSwitch.uiMaskRtStat));
//
//	ELSIF tyP0930MagConv2Btm1.tyFB.tyBtnFixedClamp.bValue = TRUE OR tyP0930MagConv2Btm1.tyFB.tyBtnRemoteClamp.bValue = TRUE
//			OR tyP0930MagConv2Btm1.tyFB.tyBtnFixedUnclamp.bValue = TRUE OR tyP0930MagConv2Btm1.tyFB.tyBtnRemoteUnclamp.bValue = TRUE
//			OR tyP0930MagConv2Btm1.tyFB.tyBtnSelUnclamp.bValue = TRUE OR tyP0930MagConv2Btm1.tyFB.tyBtnSelClamp.bValue = TRUE
//			THEN
//
//		fUIInRtStatOff(ADR(tyP0930MagConv2Btm1.tyFB.tyBtnEnt.uiMaskRtStat));
//		fUIInRtStatOff(ADR(tyP0930MagConv2Btm1.tyFB.tyBtnExit.uiMaskRtStat));
//		fUIInRtStatHide(ADR(tyP0930MagConv2Btm1.tyFB.tyBtnFixedClamp.uiMaskRtStat));
//		fUIInRtStatHide(ADR(tyP0930MagConv2Btm1.tyFB.tyBtnFixedUnclamp.uiMaskRtStat));
//		fUIInRtStatHide(ADR(tyP0930MagConv2Btm1.tyFB.tyBtnRemoteClamp.uiMaskRtStat));
//		fUIInRtStatHide(ADR(tyP0930MagConv2Btm1.tyFB.tyBtnRemoteUnclamp.uiMaskRtStat));
//		fUIInRtStatHide(ADR(tyP0930MagConv2Btm1.tyFB.tyBtnSelClamp.uiMaskRtStat));
//		fUIInRtStatHide(ADR(tyP0930MagConv2Btm1.tyFB.tyBtnSelUnclamp.uiMaskRtStat));
//		fUIInRtStatOff(ADR(tyP0930MagConv2Btm1.tyCom.tyBtnSwitch.uiMaskRtStat));
//
//	ELSE
//
//		fUIInRtStatHide(ADR(tyP0930MagConv2Btm1.tyFB.tyBtnEnt.uiMaskRtStat));
//		fUIInRtStatHide(ADR(tyP0930MagConv2Btm1.tyFB.tyBtnExit.uiMaskRtStat));
//		fUIInRtStatHide(ADR(tyP0930MagConv2Btm1.tyFB.tyBtnFixedClamp.uiMaskRtStat));
//		fUIInRtStatHide(ADR(tyP0930MagConv2Btm1.tyFB.tyBtnFixedUnclamp.uiMaskRtStat));
//		fUIInRtStatHide(ADR(tyP0930MagConv2Btm1.tyFB.tyBtnRemoteClamp.uiMaskRtStat));
//		fUIInRtStatHide(ADR(tyP0930MagConv2Btm1.tyFB.tyBtnRemoteUnclamp.uiMaskRtStat));
//		fUIInRtStatHide(ADR(tyP0930MagConv2Btm1.tyFB.tyBtnSelClamp.uiMaskRtStat));
//		fUIInRtStatHide(ADR(tyP0930MagConv2Btm1.tyFB.tyBtnSelUnclamp.uiMaskRtStat));
//		fUIInRtStatHide(ADR(tyP0930MagConv2Btm1.tyCom.tyBtnSwitch.uiMaskRtStat));
//
//	END_IF
//END_IF
//
//	IF p_tyDI.bMagConv2BtmCAB717MagSen1 THEN
//			fUIInRtStatOff(ADR(tyP0930MagConv2Btm1.tyFB.tyBtnSelClamp.uiMaskRtStat));
//	END_IF
//
//	IF p_bMagConv2Btm2Clp1ClprFixClampCtrl OR p_bMagConv2Btm2Clp1ClprRmtClampCtrl THEN
//		fUIInRtStatOff(ADR(tyP0930MagConv2Btm1.tyFB.tyBtnEnt.uiMaskRtStat));
//		fUIInRtStatOff(ADR(tyP0930MagConv2Btm1.tyFB.tyBtnExit.uiMaskRtStat));
//	END_IF
//

END_ACTION
```

#### Act_OptP0929MagConv2TopDC.st
```iecst
ACTION Act_OptP0929MagConv2TopDC:

	//Magazine Conv2eyor
	IF tyP0929MagConv2.tyTopDC.tyBtnStop.bRtCompl = TRUE THEN
		eInMagConv2Act	:= MagConvActStop;

		IF p_eInMagConv2Stat = MagConvActStop AND p_eInMagConv2Status = Done THEN
			eInMagConv2Act	:= MagConvActIdle;

			tyP0929MagConv2.tyTopDC.tyBtnStop.bRtCompl		:= FALSE;
			tyP0929MagConv2.tyTopDC.tyBtnStop.bValue		:= TRUE;
			tyP0929MagConv2.tyTopDC.tyBtnStop.bRtLk		:= TRUE;

			tyP0929MagConv2.tyTopDC.tyBtnMagIn.bRtCompl	:= FALSE;
			tyP0929MagConv2.tyTopDC.tyBtnMagIn.bValue		:= FALSE;
			tyP0929MagConv2.tyTopDC.tyBtnMagIn.bRtLk		:= FALSE;

			tyP0929MagConv2.tyTopDC.tyBtnMagOut.bRtCompl	:= FALSE;
			tyP0929MagConv2.tyTopDC.tyBtnMagOut.bValue		:= FALSE;
			tyP0929MagConv2.tyTopDC.tyBtnMagOut.bRtLk		:= FALSE;
		END_IF

	ELSIF tyP0929MagConv2.tyTopDC.tyBtnMagIn.bRtCompl = TRUE THEN
		tyP0929MagConv2.tyTopDC.tyBtnMagIn.bValue	:= TRUE;
		tyP0929MagConv2.tyTopDC.tyBtnMagIn.bRtLk	:= TRUE;

		tyP0929MagConv2.tyTopDC.tyBtnStop.bValue	:= FALSE;
		tyP0929MagConv2.tyTopDC.tyBtnStop.bRtLk	:= FALSE;

		IF p_tyNtParamCurr.eProjInMagConv2Dir = ConvDirLToR OR p_tyNtParamCurr.eProjInMagConv2Dir = ConvDirLToL THEN

			eInMagConv2Act	:= MagConvActSetMtrSigOnOrLToR;

			IF p_eInMagConv2Stat = MagConvActSetMtrSigOnOrLToR AND p_eInMagConv2Status = Done THEN
				eInMagConv2Act	:= MagConvActIdle;

				tyP0929MagConv2.tyTopDC.tyBtnMagIn.bRtCompl	:= FALSE;
			END_IF

		ELSE

			eInMagConv2Act	:= MagConvActSetMtrDirOrRToL;

			IF p_eInMagConv2Stat = MagConvActSetMtrDirOrRToL AND p_eInMagConv2Status = Done THEN
				eInMagConv2Act	:= MagConvActIdle;

				tyP0929MagConv2.tyTopDC.tyBtnMagIn.bRtCompl	:= FALSE;
			END_IF

		END_IF

	ELSIF tyP0929MagConv2.tyTopDC.tyBtnMagOut.bRtCompl = TRUE THEN
		tyP0929MagConv2.tyTopDC.tyBtnMagOut.bValue	:= TRUE;
		tyP0929MagConv2.tyTopDC.tyBtnMagOut.bRtLk	:= TRUE;

		tyP0929MagConv2.tyTopDC.tyBtnStop.bValue	:= FALSE;
		tyP0929MagConv2.tyTopDC.tyBtnStop.bRtLk	:= FALSE;

		IF p_tyNtParamCurr.eProjInMagConv2Dir = ConvDirLToR OR p_tyNtParamCurr.eProjInMagConv2Dir = ConvDirRToR THEN

			eInMagConv2Act	:= MagConvActSetMtrSigOnOrLToR;

			IF p_eInMagConv2Stat = MagConvActSetMtrSigOnOrLToR AND p_eInMagConv2Status = Done THEN
				eInMagConv2Act	:= MagConvActIdle;

				tyP0929MagConv2.tyTopDC.tyBtnMagOut.bRtCompl	:= FALSE;
			END_IF

		ELSE

			eInMagConv2Act	:= MagConvActSetMtrDirOrRToL;

			IF p_eInMagConv2Stat = MagConvActSetMtrDirOrRToL AND p_eInMagConv2Status = Done THEN
				eInMagConv2Act	:= MagConvActIdle;

				tyP0929MagConv2.tyTopDC.tyBtnMagOut.bRtCompl	:= FALSE;
			END_IF

		END_IF

	END_IF

	IF tyP0929MagConv2.tyCom.tyBtnSwitch.bValue = TRUE THEN
		//Mag Conv2 Stopper1
		IF p_bStopper1TwoCtrlOut = FALSE THEN
			IF tyP0929MagConv2.tyTopDC.tyBtnEntStprExt.bRtCompl = TRUE THEN
				tyP0929MagConv2.tyTopDC.tyBtnEntStprExt.bValue := TRUE;
				tyP0929MagConv2.tyTopDC.tyBtnEntStprRet.bValue := FALSE;

				eStopper1Act2	:= PneuActSetExt;

				IF p_eStopper1Stat2 = PneuActSetExt AND p_eStopper1Status2 = Done THEN
					eStopper1Act2	:= PneuActIdle;

					tyP0929MagConv2.tyTopDC.tyBtnEntStprExt.bRtCompl	:= FALSE;
				END_IF

			ELSIF tyP0929MagConv2.tyTopDC.tyBtnEntStprRet.bRtCompl = TRUE THEN
				tyP0929MagConv2.tyTopDC.tyBtnEntStprRet.bValue := TRUE;
				tyP0929MagConv2.tyTopDC.tyBtnEntStprExt.bValue := FALSE;

				eStopper1Act2	:= PneuActSetRet;

				IF p_eStopper1Stat2 = PneuActSetRet AND p_eStopper1Status2 = Done THEN
					eStopper1Act2	:= PneuActIdle;

					tyP0929MagConv2.tyTopDC.tyBtnEntStprRet.bRtCompl	:= FALSE;
				END_IF
			END_IF

		ELSE
			IF (tyP0929MagConv2.tyTopDC.tyBtnEntStprExt.bRtCompl = TRUE) OR (tyP0929MagConv2.tyTopDC.tyBtnEntStprRet.bRtCompl = TRUE) THEN
				IF (tyP0929MagConv2.tyTopDC.tyBtnEntStprExt.bValue = TRUE) AND (tyP0929MagConv2.tyTopDC.tyBtnEntStprRet.bValue = TRUE) THEN
					eStopper1Act2	:= PneuActSetAll;

					IF p_eStopper1Stat2 = PneuActSetAll AND p_eStopper1Status2 = Done THEN
						eStopper1Act2	:= PneuActIdle;

						tyP0929MagConv2.tyTopDC.tyBtnEntStprExt.bRtCompl		:= FALSE;
						tyP0929MagConv2.tyTopDC.tyBtnEntStprRet.bRtCompl			:= FALSE;
					END_IF
					/////////i edited the ret to ext
				ELSIF (tyP0929MagConv2.tyTopDC.tyBtnEntStprExt.bValue = TRUE) AND (tyP0929MagConv2.tyTopDC.tyBtnEntStprRet.bValue = FALSE) THEN
					eStopper1Act2	:= PneuActSetExt;(**)

					IF p_eStopper1Stat2 = PneuActSetExt (**) AND p_eStopper1Status2 = Done THEN
						eStopper1Act2	:= PneuActIdle;

						tyP0929MagConv2.tyTopDC.tyBtnEntStprExt.bRtCompl		:= FALSE;
						tyP0929MagConv2.tyTopDC.tyBtnEntStprRet.bRtCompl		:= FALSE;
					END_IF

				ELSIF (tyP0929MagConv2.tyTopDC.tyBtnEntStprExt.bValue = FALSE) AND (tyP0929MagConv2.tyTopDC.tyBtnEntStprRet.bValue = TRUE) THEN
					eStopper1Act2	:= PneuActSetRet;

					IF p_eStopper1Stat2 = PneuActSetRet AND p_eStopper1Status2 = Done THEN
						eStopper1Act2	:= PneuActIdle;

						tyP0929MagConv2.tyTopDC.tyBtnEntStprExt.bRtCompl		:= FALSE;
						tyP0929MagConv2.tyTopDC.tyBtnEntStprRet.bRtCompl			:= FALSE;
					END_IF
					///////
				ELSE
					eStopper1Act2	:= PneuActRstAll;

					IF p_eStopper1Stat2 = PneuActRstAll AND p_eStopper1Status2 = Done THEN
						eStopper1Act2	:= PneuActIdle;

						tyP0929MagConv2.tyTopDC.tyBtnEntStprExt.bRtCompl		:= FALSE;
						tyP0929MagConv2.tyTopDC.tyBtnEntStprRet.bRtCompl			:= FALSE;
					END_IF

				END_IF
			END_IF
		END_IF//stopper1

		//Mag Conv2 Stopper2
		IF p_bStopper2TwoCtrlOut = FALSE THEN
			IF tyP0929MagConv2.tyTopDC.tyBtnMidStprExt.bRtCompl = TRUE THEN
				tyP0929MagConv2.tyTopDC.tyBtnMidStprExt.bValue := TRUE;
				tyP0929MagConv2.tyTopDC.tyBtnMidStprRet.bValue := FALSE;

				eStopper2Act2	:= PneuActSetExt;

				IF p_eStopper2Stat2 = PneuActSetExt AND p_eStopper2Status2 = Done THEN
					eStopper2Act2	:= PneuActIdle;

					tyP0929MagConv2.tyTopDC.tyBtnMidStprExt.bRtCompl	:= FALSE;
				END_IF

			ELSIF tyP0929MagConv2.tyTopDC.tyBtnMidStprRet.bRtCompl = TRUE THEN
				tyP0929MagConv2.tyTopDC.tyBtnMidStprRet.bValue := TRUE;
				tyP0929MagConv2.tyTopDC.tyBtnMidStprExt.bValue := FALSE;

				eStopper2Act2	:= PneuActSetRet;

				IF p_eStopper2Stat2 = PneuActSetRet AND p_eStopper2Status2 = Done THEN
					eStopper2Act2	:= PneuActIdle;

					tyP0929MagConv2.tyTopDC.tyBtnMidStprRet.bRtCompl	:= FALSE;
				END_IF
			END_IF

		ELSE
			IF (tyP0929MagConv2.tyTopDC.tyBtnMidStprExt.bRtCompl = TRUE) OR (tyP0929MagConv2.tyTopDC.tyBtnMidStprRet.bRtCompl = TRUE) THEN
				IF (tyP0929MagConv2.tyTopDC.tyBtnMidStprExt.bValue = TRUE) AND (tyP0929MagConv2.tyTopDC.tyBtnMidStprRet.bValue = TRUE) THEN
					eStopper2Act2	:= PneuActSetAll;

					IF p_eStopper2Stat2 = PneuActSetAll AND p_eStopper2Status2 = Done THEN
						eStopper2Act2	:= PneuActIdle;

						tyP0929MagConv2.tyTopDC.tyBtnMidStprExt.bRtCompl		:= FALSE;
						tyP0929MagConv2.tyTopDC.tyBtnMidStprRet.bRtCompl			:= FALSE;
					END_IF
					/////////i edited the ret to ext
				ELSIF (tyP0929MagConv2.tyTopDC.tyBtnMidStprExt.bValue = TRUE) AND (tyP0929MagConv2.tyTopDC.tyBtnMidStprRet.bValue = FALSE) THEN
					eStopper2Act2	:= PneuActSetExt;(**)

					IF p_eStopper2Stat2 = PneuActSetExt (**) AND p_eStopper2Status2 = Done THEN
						eStopper2Act2	:= PneuActIdle;

						tyP0929MagConv2.tyTopDC.tyBtnMidStprExt.bRtCompl		:= FALSE;
						tyP0929MagConv2.tyTopDC.tyBtnMidStprRet.bRtCompl		:= FALSE;
					END_IF

				ELSIF (tyP0929MagConv2.tyTopDC.tyBtnMidStprExt.bValue = FALSE) AND (tyP0929MagConv2.tyTopDC.tyBtnMidStprRet.bValue = TRUE) THEN
					eStopper2Act2	:= PneuActSetRet;

					IF p_eStopper2Stat2 = PneuActSetRet AND p_eStopper2Status2 = Done THEN
						eStopper2Act2	:= PneuActIdle;

						tyP0929MagConv2.tyTopDC.tyBtnMidStprExt.bRtCompl		:= FALSE;
						tyP0929MagConv2.tyTopDC.tyBtnMidStprRet.bRtCompl			:= FALSE;
					END_IF
					///////
				ELSE
					eStopper2Act2	:= PneuActRstAll;

					IF p_eStopper2Stat2 = PneuActRstAll AND p_eStopper2Status2 = Done THEN
						eStopper2Act2	:= PneuActIdle;

						tyP0929MagConv2.tyTopDC.tyBtnMidStprExt.bRtCompl		:= FALSE;
						tyP0929MagConv2.tyTopDC.tyBtnMidStprRet.bRtCompl			:= FALSE;
					END_IF

				END_IF
			END_IF
		END_IF//stopper2

		//Mag Conv2 Stopper3
		IF p_bStopper3TwoCtrlOut = FALSE THEN
			IF tyP0929MagConv2.tyTopDC.tyBtnExtStprExt.bRtCompl = TRUE THEN
				tyP0929MagConv2.tyTopDC.tyBtnExtStprExt.bValue := TRUE;
				tyP0929MagConv2.tyTopDC.tyBtnExtStprRet.bValue := FALSE;

				eStopper3Act2	:= PneuActSetExt;

				IF p_eStopper3Stat2 = PneuActSetExt AND p_eStopper3Status2 = Done THEN
					eStopper3Act2	:= PneuActIdle;

					tyP0929MagConv2.tyTopDC.tyBtnExtStprExt.bRtCompl	:= FALSE;
				END_IF

			ELSIF tyP0929MagConv2.tyTopDC.tyBtnExtStprRet.bRtCompl = TRUE THEN
				tyP0929MagConv2.tyTopDC.tyBtnExtStprRet.bValue := TRUE;
				tyP0929MagConv2.tyTopDC.tyBtnExtStprExt.bValue := FALSE;

				eStopper3Act2	:= PneuActSetRet;

				IF p_eStopper3Stat2 = PneuActSetRet AND p_eStopper3Status2 = Done THEN
					eStopper3Act2	:= PneuActIdle;

					tyP0929MagConv2.tyTopDC.tyBtnExtStprRet.bRtCompl	:= FALSE;
				END_IF
			END_IF

		ELSE
			IF (tyP0929MagConv2.tyTopDC.tyBtnExtStprExt.bRtCompl = TRUE) OR (tyP0929MagConv2.tyTopDC.tyBtnExtStprRet.bRtCompl = TRUE) THEN
				IF (tyP0929MagConv2.tyTopDC.tyBtnExtStprExt.bValue = TRUE) AND (tyP0929MagConv2.tyTopDC.tyBtnExtStprRet.bValue = TRUE) THEN
					eStopper3Act2	:= PneuActSetAll;

					IF p_eStopper3Stat2 = PneuActSetAll AND p_eStopper3Status2 = Done THEN
						eStopper3Act2	:= PneuActIdle;

						tyP0929MagConv2.tyTopDC.tyBtnExtStprExt.bRtCompl		:= FALSE;
						tyP0929MagConv2.tyTopDC.tyBtnExtStprRet.bRtCompl			:= FALSE;
					END_IF
					/////////i edited the ret to ext
				ELSIF (tyP0929MagConv2.tyTopDC.tyBtnExtStprExt.bValue = TRUE) AND (tyP0929MagConv2.tyTopDC.tyBtnExtStprRet.bValue = FALSE) THEN
					eStopper3Act2	:= PneuActSetExt;(**)

					IF p_eStopper3Stat2 = PneuActSetExt (**) AND p_eStopper3Status2 = Done THEN
						eStopper3Act2	:= PneuActIdle;

						tyP0929MagConv2.tyTopDC.tyBtnExtStprExt.bRtCompl		:= FALSE;
						tyP0929MagConv2.tyTopDC.tyBtnExtStprRet.bRtCompl		:= FALSE;
					END_IF

				ELSIF (tyP0929MagConv2.tyTopDC.tyBtnExtStprExt.bValue = FALSE) AND (tyP0929MagConv2.tyTopDC.tyBtnExtStprRet.bValue = TRUE) THEN
					eStopper3Act2	:= PneuActSetRet;

					IF p_eStopper3Stat2 = PneuActSetRet AND p_eStopper3Status2 = Done THEN
						eStopper3Act2	:= PneuActIdle;

						tyP0929MagConv2.tyTopDC.tyBtnExtStprExt.bRtCompl		:= FALSE;
						tyP0929MagConv2.tyTopDC.tyBtnExtStprRet.bRtCompl			:= FALSE;
					END_IF
					///////
				ELSE
					eStopper3Act2	:= PneuActRstAll;

					IF p_eStopper3Stat2 = PneuActRstAll AND p_eStopper3Status2 = Done THEN
						eStopper3Act2	:= PneuActIdle;

						tyP0929MagConv2.tyTopDC.tyBtnExtStprExt.bRtCompl		:= FALSE;
						tyP0929MagConv2.tyTopDC.tyBtnExtStprRet.bRtCompl			:= FALSE;
					END_IF

				END_IF
			END_IF
		END_IF//stopper3

		//ent
		tyP0929MagConv2.tyTopFB.tyBtnEntStprExt.bRtCompl		:= FALSE;
		tyP0929MagConv2.tyTopFB.tyBtnEntStprExt.bValue		:= FALSE;
		tyP0929MagConv2.tyTopFB.tyBtnEntStprRet.bRtCompl		:= FALSE;
		tyP0929MagConv2.tyTopFB.tyBtnEntStprRet.bValue		:= FALSE;

		//mid
		tyP0929MagConv2.tyTopFB.tyBtnMidStprExt.bRtCompl		:= FALSE;
		tyP0929MagConv2.tyTopFB.tyBtnMidStprExt.bValue		:= FALSE;
		tyP0929MagConv2.tyTopFB.tyBtnMidStprRet.bRtCompl		:= FALSE;
		tyP0929MagConv2.tyTopFB.tyBtnMidStprRet.bValue		:= FALSE;

		//ext
		tyP0929MagConv2.tyTopFB.tyBtnExtStprExt.bRtCompl		:= FALSE;
		tyP0929MagConv2.tyTopFB.tyBtnExtStprExt.bValue		:= FALSE;
		tyP0929MagConv2.tyTopFB.tyBtnExtStprRet.bRtCompl		:= FALSE;
		tyP0929MagConv2.tyTopFB.tyBtnExtStprRet.bValue		:= FALSE;
	END_IF

	//Mask
//	IF p_eInMagConv2Status = Error THEN
//
//		fUIInRtStatOff(ADR(tyP0929MagConv2.tyTopDC.tyBtnMagIn.uiMaskRtStat));
//		fUIInRtStatOff(ADR(tyP0929MagConv2.tyTopDC.tyBtnMagOut.uiMaskRtStat));
//		fUIInRtStatOff(ADR(tyP0929MagConv2.tyTopDC.tyBtnFixedClamp.uiMaskRtStat));
//		fUIInRtStatOff(ADR(tyP0929MagConv2.tyTopDC.tyBtnFixedUnclamp.uiMaskRtStat));
//		fUIInRtStatOff(ADR(tyP0929MagConv2.tyTopDC.tyBtnRemoteClamp.uiMaskRtStat));
//		fUIInRtStatOff(ADR(tyP0929MagConv2.tyTopDC.tyBtnRemoteUnclamp.uiMaskRtStat));
//		fUIInRtStatOff(ADR(tyP0929MagConv2.tyTopDC.tyBtnSelClamp.uiMaskRtStat));
//		fUIInRtStatOff(ADR(tyP0929MagConv2.tyTopDC.tyBtnSelUnclamp.uiMaskRtStat));
//
//	ELSIF tyP0929MagConv2.tyTopDC.tyBtnMagIn.bValue = TRUE THEN
//
//		fUIInRtStatHide(ADR(tyP0929MagConv2.tyTopDC.tyBtnMagIn.uiMaskRtStat));
//		fUIInRtStatOff(ADR(tyP0929MagConv2.tyTopDC.tyBtnMagOut.uiMaskRtStat));
//		fUIInRtStatOff(ADR(tyP0929MagConv2.tyTopDC.tyBtnFixedClamp.uiMaskRtStat));
//		fUIInRtStatOff(ADR(tyP0929MagConv2.tyTopDC.tyBtnFixedUnclamp.uiMaskRtStat));
//		fUIInRtStatOff(ADR(tyP0929MagConv2.tyTopDC.tyBtnRemoteClamp.uiMaskRtStat));
//		fUIInRtStatOff(ADR(tyP0929MagConv2.tyTopDC.tyBtnRemoteUnclamp.uiMaskRtStat));
//		fUIInRtStatOff(ADR(tyP0929MagConv2.tyTopDC.tyBtnSelClamp.uiMaskRtStat));
//		fUIInRtStatOff(ADR(tyP0929MagConv2.tyTopDC.tyBtnSelUnclamp.uiMaskRtStat));
//
//	ELSIF tyP0929MagConv2.tyTopDC.tyBtnMagOut.bValue = TRUE THEN
//
//		fUIInRtStatOff(ADR(tyP0929MagConv2.tyTopDC.tyBtnMagIn.uiMaskRtStat));
//		fUIInRtStatHide(ADR(tyP0929MagConv2.tyTopDC.tyBtnMagOut.uiMaskRtStat));
//		fUIInRtStatOff(ADR(tyP0929MagConv2.tyTopDC.tyBtnFixedClamp.uiMaskRtStat));
//		fUIInRtStatOff(ADR(tyP0929MagConv2.tyTopDC.tyBtnFixedUnclamp.uiMaskRtStat));
//		fUIInRtStatOff(ADR(tyP0929MagConv2.tyTopDC.tyBtnRemoteClamp.uiMaskRtStat));
//		fUIInRtStatOff(ADR(tyP0929MagConv2.tyTopDC.tyBtnRemoteUnclamp.uiMaskRtStat));
//		fUIInRtStatOff(ADR(tyP0929MagConv2.tyTopDC.tyBtnSelClamp.uiMaskRtStat));
//		fUIInRtStatOff(ADR(tyP0929MagConv2.tyTopDC.tyBtnSelUnclamp.uiMaskRtStat));
//
//	ELSE
//
//		fUIInRtStatHide(ADR(tyP0929MagConv2.tyTopDC.tyBtnMagIn.uiMaskRtStat));
//		fUIInRtStatHide(ADR(tyP0929MagConv2.tyTopDC.tyBtnMagOut.uiMaskRtStat));
//		fUIInRtStatHide(ADR(tyP0929MagConv2.tyTopDC.tyBtnFixedClamp.uiMaskRtStat));
//		fUIInRtStatHide(ADR(tyP0929MagConv2.tyTopDC.tyBtnFixedUnclamp.uiMaskRtStat));
//		fUIInRtStatHide(ADR(tyP0929MagConv2.tyTopDC.tyBtnRemoteClamp.uiMaskRtStat));
//		fUIInRtStatHide(ADR(tyP0929MagConv2.tyTopDC.tyBtnRemoteUnclamp.uiMaskRtStat));
//		fUIInRtStatHide(ADR(tyP0929MagConv2.tyTopDC.tyBtnSelClamp.uiMaskRtStat));
//		fUIInRtStatHide(ADR(tyP0929MagConv2.tyTopDC.tyBtnSelUnclamp.uiMaskRtStat));
//
//	END_IF
//

END_ACTION
```
